F_ConfigPositionEmulation_002();

END_FUNCTION

// ---- 10_Project/11_Emu/10_Config/F_ConfigPositionEmulation_001.TcPOU
FUNCTION F_ConfigPositionEmulation_001








(****************************** 10-001-0201-01-0 ************************************)
(**************************** LowLift Unit Emulation ***************************)
// Configuration emulation
fbF_10_001_0201_01_0_Emulation.Config.Position_Max_Down			:= 0;
fbF_10_001_0201_01_0_Emulation.Config.Position_Max_Up	  			:= 600;	
fbF_10_001_0201_01_0_Emulation.Config.Position_Down				:= 100;
fbF_10_001_0201_01_0_Emulation.Config.Position_Up	  				:= 500;






(****************************** 10-001-0203-02-0 ************************************)
(******************************** Profile Check Emulation *****************************)
// Configuration emulation
fbF_10_001_0203_02_0_Emulation.Config.DefaultWidth					:= 800;
fbF_10_001_0203_02_0_Emulation.Config.DefaultLength					:= 1200;	

(****************************** 10-001-0203-03-0 ************************************)
// Configuration Scanner emulation
fbF_10_001_0203_03_0_Emulation.Config.CreateLabelLength				:= 18; // Label length when ATQ Msg field data is set to 'CREATECODE'







(****************************** 10-001-0204-01-0 ************************************)
(**************************** TurnTable with one drive ***************************)
// Configuration emulation
fbF_10_001_0204_01_0_Emulation.Config.TurnTableCfg.Position_Max_CW	  	:= 500;
fbF_10_001_0204_01_0_Emulation.Config.TurnTableCfg.Position_Max_CCW	:= 0;	
fbF_10_001_0204_01_0_Emulation.Config.TurnTableCfg.Position_CW	  		:= 400;
fbF_10_001_0204_01_0_Emulation.Config.TurnTableCfg.Position_CCW		:= 0;
fbF_10_001_0204_01_0_Emulation.Config.TurnTableCfg.Position_Middle_CW	:= 200;
fbF_10_001_0204_01_0_Emulation.Config.TurnTableCfg.Position_Middle_CCW	:= 200;






(****************************** 10-001-0207-02-0 ************************************)
(****************************** PalletMagazine Addon *************************************)

fbF_10_001_0207_02_0_Emulation.Config.MaxLiftPosition			:= 600;
fbF_10_001_0207_02_0_Emulation.Config.NumberPalletStack		:= 5;	
fbF_10_001_0207_02_0_Emulation.Config.NumberPalletFull			:= 7;






(****************************** 10-001-0209-01-0 ************************************)
(**************************** Transfer Unit Emulation ***************************)
// Configuration emulation
fbF_10_001_0209_01_0_Emulation.Config.Position_Max_Down			:= 0;
fbF_10_001_0209_01_0_Emulation.Config.Position_Max_Up	  			:= 400;	
fbF_10_001_0209_01_0_Emulation.Config.Position_Down				:= 100;
fbF_10_001_0209_01_0_Emulation.Config.Position_Up	  				:= 300;






(****************************** 10-001-0212-01-0 ************************************)
(**************************** Transfer Unit Emulation ***************************)
// Configuration emulation
fbF_10_001_0212_01_0_Emulation.Config.Position_Max_Down			:= 0;
fbF_10_001_0212_01_0_Emulation.Config.Position_Max_Up	  			:= 400;	
fbF_10_001_0212_01_0_Emulation.Config.Position_Down				:= 100;
fbF_10_001_0212_01_0_Emulation.Config.Position_Up	  				:= 300;



(****************************** 10-001-0213-02-0 ************************************)
(****************************** PalletMagazine Addon *************************************)

fbF_10_001_0213_02_0_Emulation.Config.MaxLiftPosition			:= 600;
fbF_10_001_0213_02_0_Emulation.Config.NumberPalletStack		:= 5;	
fbF_10_001_0213_02_0_Emulation.Config.NumberPalletFull			:= 7;





















(****************************** 10-001-0221-01-0 ************************************)
(**************************** Transfer Unit Emulation ***************************)
// Configuration emulation
fbF_10_001_0221_01_0_Emulation.Config.Position_Max_Down			:= 0;
fbF_10_001_0221_01_0_Emulation.Config.Position_Max_Up	  			:= 400;	
fbF_10_001_0221_01_0_Emulation.Config.Position_Down				:= 100;
fbF_10_001_0221_01_0_Emulation.Config.Position_Up	  				:= 300;




(****************************** 10-001-0222-01-0 ************************************)
(**************************** Transfer Unit Emulation ***************************)
// Configuration emulation
fbF_10_001_0222_01_0_Emulation.Config.Position_Max_Down			:= 0;
fbF_10_001_0222_01_0_Emulation.Config.Position_Max_Up	  			:= 400;	
fbF_10_001_0222_01_0_Emulation.Config.Position_Down				:= 100;
fbF_10_001_0222_01_0_Emulation.Config.Position_Up	  				:= 300;










(****************************** 10-001-0230-01-0 ************************************)
(**************************** TransferCC Emulation ***************************)
// Configuration emulation
fbF_10_001_0230_01_0_Emulation.Config.Position_Max_Left			:= 0;
fbF_10_001_0230_01_0_Emulation.Config.Position_Max_Right	  			:= 600;	
fbF_10_001_0230_01_0_Emulation.Config.Position_Left				:= 100;
fbF_10_001_0230_01_0_Emulation.Config.Position_Right	  				:= 500;

END_FUNCTION

// ---- 10_Project/11_Emu/10_Config/F_ConfigPositionEmulation_002.TcPOU
FUNCTION F_ConfigPositionEmulation_002

END_FUNCTION

// ---- 10_Project/11_Emu/10_Config/F_ConfigGroupEmulation.TcPOU
FUNCTION F_ConfigGroupEmulation




(********************************* Group *************************************
 Switching Group  
**********************************************************************************)
fbSG_001_Emulation.Config.Autostart := TRUE;


(********************************* Group *************************************
 Switching Group  
**********************************************************************************)
fbSG_002_Emulation.Config.Autostart := TRUE;

END_FUNCTION

// ---- 10_Project/11_Emu/10_Config/F_ConfigSubSystemEmulation.TcPOU
FUNCTION F_ConfigSubSystemEmulation : BOOL

;

END_FUNCTION

// ---- 10_Project/10_App/11_Custom/F_DebugCompositionCustomization.TcPOU
FUNCTION F_DebugCompositionCustomization : BOOL



(****************************************************************************************
   Add custom code that shall be executed during debug here.
*****************************************************************************************)
;


(****************************************************************************************
   Example: Configure project when running Demo3D simulator
*****************************************************************************************)
IF(DEMO3D_SIM_ENABLED) THEN
	;
	(*
	Groups.fbSG_001.HW_Inputs.AutoOnPB 						:= TRUE;
	Groups.fbSG_001.HW_Inputs.EmergencyCircuitOK 			:= TRUE;
	Groups.fbSG_001.HW_Inputs.ManAutoSW 					:= TRUE;
	Groups.fbSG_001.HW_Inputs.ResetErrorPB 					:= ResetErrorSG1; 
	Groups.fbSG_001.HW_Inputs.MainContactorOFF				:= TRUE; 
	Groups.fbSG_001.HW_Inputs.FeedbackMainContactorOFF[1]	:= TRUE; 
	Groups.fbSG_001.HW_Inputs.FeedbackMainContactorOFF[2]	:= TRUE; 
	Groups.fbSG_001.HW_Inputs.FeedbackMainContactorOFF[3]	:= TRUE; 
	Groups.fbSG_001.HW_Inputs.FeedbackMainContactorOFF[4]	:= TRUE; 
	Groups.fbSG_001.HW_Inputs.FireAlarm						:= TRUE; 
	*)
END_IF

END_FUNCTION

// ---- 20_Product/20_ProBox/22_ProMove/14_Groups/10_App/FB_ProBOXSG.TcPOU
FUNCTION_BLOCK FB_ProBOXSG EXTENDS FB_GroupConv
(**************************************************************************************
 * 	Application		:	BoxControl Framework
 *	Revision		:	$$
 *	Revision date	:	$$
 *	Last changed by	:	$$
 *	URL				:	$$
 *
 *	Purpose			:	ProBox Switching group - Controls a group of elements.
 *
 * ------------------------------------------------------------------------------------
 *	Copyright Swisslog [IP AG], Switzerland. All rights reserved.
 * 
 * ------------------------------------------------------------------------------------
 *	
 * 	Revision History: 
 *
 * 	VERSION			DATE			INITIALS			DESCRIPTION 
 **************************************************************************************)
VAR_INPUT
	HW_Inputs				: ST_HW_InputsSG_ProBOX; // HW-Inputs 
	Config					: ST_CFG_ProBOXSG; // Configuration 
	LocalStopCmd			: BOOL; // Stopping cmd
END_VAR

VAR_OUTPUT
	HW_Outputs				: ST_HW_OutputsSG_ProBOX; // HW-Outputs
	CtrlOut					: ST_CtlrOutProBoxSG; // Summary of input commands from Operator panel(s)
END_VAR

VAR
	ProBoxSG_CFG			: ST_CFG_ProBoxSG;
	Inputs					: ST_SG_Inputs_ProBOX; // Module internal inputs
	Outputs					: ST_SG_Outputs_ProBOX; // Module Internal outputs
	ResetFlag				: BOOL; // Flag to detect reset pulse
	PendingElementError		: BOOL; // An member element is in error state
	fbStartingDelay			: TON; // Timer for startup delay 
	fbForcedStopDelay		: TON; // Timer for forcing a group to stop
	fbResetPulse			: TOF; // Timer for a longer reset pulse
	fbTrigReset				: R_TRIG; // Reset positive flag
	i						: INT;
	ManualModeDelayCnt		: INT; //Delay the Manual Mode  a few cycle in order to send GSR with correct stopped state
END_VAR

VAR PERSISTENT
	Settings				: ST_CFG_ProBoxSG; // Settings - Active configuration
END_VAR

(**************************************************************************************************************
   Input mapping
***************************************************************************************************************)
A_InputMapping();


(**************************************************************************************************************
   Initialization
***************************************************************************************************************)
A_Init();


(**************************************************************************************************************
   Monitoring input signals
***************************************************************************************************************)
A_SignalMonitoring();

//Process Emergency State signal
_M_ProcessEmgState();


(**************************************************************************************************************
   Errorhandler
***************************************************************************************************************)
A_ErrorHandler();


(**************************************************************************************************************
  Mode control
***************************************************************************************************************)
A_ModeControl();


(**************************************************************************************************************
  State control
***************************************************************************************************************)
A_StateControl();


(**************************************************************************************************************
   InterfaceHandlerOut
***************************************************************************************************************)
A_InterfaceHandlerOut();
	

(**************************************************************************************************************
   Output mapping
***************************************************************************************************************)	
A_OutputMapping();

METHOD PRIVATE _M_ProcessEmgState : BOOL
VAR_INST
	InternalStopPending 	: BOOL :=TRUE; //has internal error memory flag
	fbBlink_ExternalStop	: FB_GeneratePulse := (Start := TRUE, PulseTimeOn := T#1S, PulseTimeOff := T#2S); // On 1 sec, off 2 sec
END_VAR
VAR
	InternalStop	: BOOL;
	ExternalStop	: BOOL;
	LampState		: BOOL; //Lamp State
	EmgOk			: BOOL := FALSE;
END_VAR
InternalStop := NOT Inputs.States.EmgStatus.eInternal OR Inputs.States.EmgStatus.eInternError;
ExternalStop := NOT Inputs.States.EmgStatus.eExternal;

IF(NOT GroupData.Init) THEN
	InternalStopPending:=FALSE;
END_IF

//EMG STOP
IF(ExternalStop OR InternalStop) THEN			
	//Internal emg stop is no longer active, but External (safety zone is not acknowledged)	
	IF(ExternalStop AND InternalStopPending AND NOT InternalStop) THEN
		LampState := System.fbBlink_500ms.Pulse;	
	// IF External stop but internal (AK group) is ok
	ELSIF(ExternalStop AND NOT InternalStop) THEN
		fbBlink_ExternalStop();
		LampState := fbBlink_ExternalStop.Pulse;
	ELSE
		LampState := TRUE;
		InternalStopPending := InternalStop; //Set Mem flag
	END_IF

ELSE	
	LampState := FALSE;
	InternalStopPending := FALSE;
	EmgOk:=TRUE;
END_IF


Inputs.States.EmergencyCircuitOK := EmgOk;
Outputs.EmgStopStatus := _M_ProcessEmgState := LampState;
END_METHOD

METHOD PRIVATE _M_ProcessInputs

VAR
	i,j:INT;
	iMax:INT;
END_VAR
	 
//process inputs and create summary
//AK
	Inputs.OpSummary.OpAutoOn		:= HW_Inputs.AK.OpAutoOn;
	Inputs.OpSummary.OpManAuto		:= HW_Inputs.AK.OpManAuto; //NC
	Inputs.OpSummary.OpMcOff 		:= HW_Inputs.AK.OpMcOff; //NC
	Inputs.OpSummary.OpMcOn 		:= HW_Inputs.AK.OpMcOn;
	Inputs.OpSummary.OpResetError	:= HW_Inputs.AK.OpResetError;
	Inputs.OpSummary.OpResetSafety	:= HW_Inputs.AK.OpResetSafety;	
	Inputs.OpSummary.OpEntryReq   	:= HW_Inputs.AK.OpEntryReq; //NC //Hi=Auto, low=Entry
	Inputs.OpSummary.OpEmgDrive   	:= HW_Inputs.AK.OpEmgDrive AND HW_Inputs.AK.OpManAuto = FALSE; (* and Manual mode*)
	FOR j:=1 TO 2 DO
		Inputs.OpSummary.Conv[j].OpDriveCvFwd := HW_Inputs.AK.Conv[j].OpDriveCvFwd AND HW_Inputs.AK.OpManAuto = FALSE; (*Manual mode*) 
		Inputs.OpSummary.Conv[j].OpDriveCvRev := HW_Inputs.AK.Conv[j].OpDriveCvRev AND HW_Inputs.AK.OpManAuto = FALSE; (*Manual mode*)		
		Inputs.OpSummary.Conv[j].OpMovePos 	  := HW_Inputs.AK.Conv[j].OpMovePos    AND HW_Inputs.AK.OpManAuto = FALSE; (*Manual mode*)
		Inputs.OpSummary.Conv[j].OpMoveNeg    := HW_Inputs.AK.Conv[j].OpMoveNeg    AND HW_Inputs.AK.OpManAuto = FALSE; (*Manual mode*)
	END_FOR	
	



//AP
	iMax :=SEL(Settings.NumberOfAPs<GVL_PB_SG.NUMBER_OF_AP_PANELS, GVL_PB_SG.NUMBER_OF_AP_PANELS, Settings.NumberOfAPs);
	FOR i:=1 TO iMax DO 
		Inputs.OpSummary.OpAutoOn		:= Inputs.OpSummary.OpAutoOn 		OR HW_Inputs.AP[i].OpAutoOn;
		Inputs.OpSummary.OpManAuto		:= Inputs.OpSummary.OpManAuto 		AND HW_Inputs.AP[i].OpManAuto; //NC
		Inputs.OpSummary.OpMcOff 		:= Inputs.OpSummary.OpMcOff 		AND HW_Inputs.AP[i].OpMcOff; //NC
		Inputs.OpSummary.OpMcOn 		:= Inputs.OpSummary.OpMcOn			OR HW_Inputs.AP[i].OpMcOn;
		Inputs.OpSummary.OpResetError	:= Inputs.OpSummary.OpResetError 	OR HW_Inputs.AP[i].OpResetError;
		Inputs.OpSummary.OpResetSafety  := Inputs.OpSummary.OpResetSafety 	OR HW_Inputs.AP[i].OpResetSafety;		
		Inputs.OpSummary.OpEntryReq     := Inputs.OpSummary.OpEntryReq     AND HW_Inputs.AP[i].OpEntryReq; //NC, Hi=Auto, low=Entry
		Inputs.OpSummary.OpEmgDrive     := Inputs.OpSummary.OpEmgDrive     OR (HW_Inputs.AP[i].OpEmgDrive    AND HW_Inputs.AP[i].OpManAuto = FALSE); (*Manual mode*)
		// manual controls of the carriage only allowed if switch is in manual mode
		FOR j:=1 TO 2 DO		 
			Inputs.OpSummary.Conv[j].OpDriveCvFwd := Inputs.OpSummary.Conv[j].OpDriveCvFwd OR (HW_Inputs.AP[i].Conv[j].OpDriveCvFwd AND HW_Inputs.AP[i].OpManAuto = FALSE); (*Manual mode*)
			Inputs.OpSummary.Conv[j].OpDriveCvRev := Inputs.OpSummary.Conv[j].OpDriveCvRev OR (HW_Inputs.AP[i].Conv[j].OpDriveCvRev AND HW_Inputs.AP[i].OpManAuto = FALSE); (*Manual mode*)
			Inputs.OpSummary.Conv[j].OpMovePos    := Inputs.OpSummary.Conv[j].OpMovePos    OR (HW_Inputs.AP[i].Conv[j].OpMovePos    AND HW_Inputs.AP[i].OpManAuto = FALSE); (*Manual mode*)
			Inputs.OpSummary.Conv[j].OpMoveNeg    := Inputs.OpSummary.Conv[j].OpMoveNeg    OR (HW_Inputs.AP[i].Conv[j].OpMoveNeg    AND HW_Inputs.AP[i].OpManAuto = FALSE); (*Manual mode*)
		END_FOR	
		
	END_FOR
END_METHOD

ACTION A_ErrorHandler:
(**************************************************************************************
 * 	NAME		A_ErrorHandling
 * 	FUNCTION	Handles group or member errors
 **************************************************************************************)
 

(**************************************************************************************************************
  Monitor group errors
***************************************************************************************************************)
M_MonitorGroupErrors();


(**************************************************************************************************************
  Input group reset
***************************************************************************************************************)

// Reset command
IF Inputs.Command.ResetErrorPB AND NOT ResetFlag THEN
	
	// If a group reset has to reset member elements as well
	IF Settings.ResetMemberElements THEN	

		// Forward reset to memeber elements
		fbGroupManager.M_ResetMemberElements(SettingsGroup.eGroupNumber);
	END_IF
		
	// Reset group itself
	GroupData.ErrorData.Error.ResetError := TRUE;
	
	// Save flag
	ResetFlag := TRUE;
	
// Reset command released
ELSIF NOT Inputs.Command.ResetErrorPB THEN
	// Reset flag
	ResetFlag := FALSE;
END_IF
END_ACTION

ACTION A_Init:
(**************************************************************************************
 * 	NAME		A_Init
 * 	FUNCTION	Initialize Group
 **************************************************************************************)

// Update Registry
M_UpdateRegistry();
 
// Set init flag after one cycle
IF NOT GroupData.Init AND GroupData.InitRunning THEN
	// When subsystem is started and initialization is allowed
	IF GroupData.OperationState.Info.SystemReady AND 
	   SettingsGroup.eGroupNumber < GroupData.OperationState.InitRelease.eLimitGroup THEN
	   
		IF M_InitGroup(FALSE) THEN
			// Group initialized - and initialization done
			GroupData.Init := TRUE;
			GroupData.InitRunning := FALSE;
			
			// Set reset cmd
			GroupData.ErrorData.Error.ResetError := TRUE;
			
			DebugMsg := CONCAT('Initialization done. Group: ', ConfigGroup.GroupName);
			fbDebugMsg.M_SendInfoMsg(DebugMsg);
		END_IF
	END_IF
// If the group is not initialized
ELSIF NOT GroupData.Init THEN
	
	// Reset internal variables
	ResetFlag := FALSE;
	PendingElementError := FALSE;
	fbStartingDelay(IN := FALSE);
	fbForcedStopDelay(IN := FALSE);
	GroupData.OperationState := GroupBase.OperationStateEmpty;
	ITC.Commands.Start := FALSE;
	ITC.Commands.Stop := FALSE;
	ITC.Commands.eMode := E_PositionMode.UNKNOWN_MODE;
	
	// Load group specific configuration to settings
	Settings := Config;
	
	// Reset values and load config
	M_PreInit();
	GroupData.InitRunning := SettingsGroup.eGroupNumber > 0;
END_IF
END_ACTION

ACTION A_InputMapping:
(**************************************************************************************
 * 	NAME		A_InputMapping
 * 	FUNCTION	Input mapping
 **************************************************************************************)
 
 
(**************************************************************************************************************
   Hardware Inputs
***************************************************************************************************************)

//Summarize inputs and set Inputs.OpSummary
_M_ProcessInputs();

// Mode
Inputs.Command.AutoMode   			:= Inputs.OpSummary.OpManAuto;//HW_Inputs.ManAutoSW;
Inputs.Command.ManualMode 			:= NOT Inputs.OpSummary.OpManAuto;

// Control
Inputs.Command.StartPB 				:=Inputs.OpSummary.OpAutoOn; //HW_Inputs.AutoOnPB;
Inputs.Command.StopPB  				:= FALSE;
Inputs.Command.ResetErrorPB			:= Inputs.OpSummary.OpResetError; //HW_Inputs.ResetErrorPB;
Inputs.Command.ResetEmgPB			:= Inputs.OpSummary.OpResetSafety; //HW_Inputs.ResetEmgergencyPB;

// Signal states							   
//Inputs.States.EmergencyCircuitOK 	:= HW_Inputs.EmergencyCircuitOK;

	// Fire alarm
IF Settings.FireAlarmUsed THEN 
	Inputs.States.FireAlarm				:= NOT HW_Inputs.Diag.FireAlarm;
ELSE Inputs.States.FireAlarm			:= FALSE;
END_IF
	
	// Checks all connected Main Contactor feedback							   
FOR i := 1 TO Settings.NumberOfContactors DO
	IF HW_Inputs.Diag.FeedbackMainContactorOFF[i] THEN
		Inputs.States.MainContactorOFF :=TRUE;
		EXIT;
	ELSE
		Inputs.States.MainContactorOFF :=FALSE;
	END_IF
END_FOR

//Inputs.States.MainContactorOFF   	:= HW_Inputs.MainContactorOFF[K.NumberOfContactors];								   

(**************************************************************************************************************
   SubsystemManager states
***************************************************************************************************************)
// Get Subsystem state
M_GetSubsystemStates();

(**************************************************************************************************************
   GroupManager
***************************************************************************************************************)

// Get group member state
Inputs.GroupMemberState 			:= fbGroupManager.M_GetGroupMemberState(SettingsGroup.eGroupNumber);
END_ACTION

ACTION A_InterfaceHandlerOut:
(**************************************************************************************
 * 	NAME		A_InterfaceHandlerOut
 * 	FUNCTION	Handle outgoing interfaces
 **************************************************************************************)
 
 
 (**************************************************************************************************************
   ITC Handler Out
***************************************************************************************************************)
M_ITC_ProcessOut();
END_ACTION

ACTION A_ModeControl:
(**************************************************************************************
 * 	NAME		A_ModeControl
 * 	FUNCTION	Handle group modes
 **************************************************************************************)
 
// Group mode
CASE GroupData.OperationState.eMode OF

	(*******************************************************************************
	  Mode: Unknown 
	********************************************************************************)
	E_PositionMode.UNKNOWN_MODE:
	
		// Group mode is default Off
		GroupData.OperationState.eMode 		:= E_PositionMode.OFF_MODE;

	(*******************************************************************************
	  Mode: OFF
	********************************************************************************)
	E_PositionMode.OFF_MODE:
	
		// If manual mode is set
		IF Inputs.Command.ManualMode THEN
			// Switch to manual mode
			GroupData.OperationState.eMode := E_PositionMode.MANUAL_MODE;
			
		// If semi auto mode is set
		ELSIF Inputs.Command.SemiAutoMode THEN
			// Switch to semi auto mode
			GroupData.OperationState.eMode := E_PositionMode.SEMI_AUTO;
			
		// If auto mode is set
		ELSIF Inputs.Command.AutoMode THEN
			// Switch to auto mode
			GroupData.OperationState.eMode := E_PositionMode.AUTO_MODE;
		END_IF

	(*******************************************************************************
	  Mode: Manual
	********************************************************************************)
	E_PositionMode.MANUAL_MODE:
	
		// If manual - stay
		IF Inputs.Command.ManualMode THEN
			;
		// If semi auto mode is set
		ELSIF Inputs.Command.SemiAutoMode THEN
			// Switch to semi auto mode
			GroupData.OperationState.eMode := E_PositionMode.SEMI_AUTO;
			
			// Send status report
			ITC.Commands.StatusReport := TRUE;
		
		// If auto is set
		ELSIF Inputs.Command.AutoMode THEN
			// Switch mode to "Auto"
			GroupData.OperationState.eMode := E_PositionMode.AUTO_MODE;
			
			// Send status report
			ITC.Commands.StatusReport := TRUE;
		ELSE
			// Switch group off
			GroupData.OperationState.eMode := E_PositionMode.OFF_MODE;
			
			// Send status report
			ITC.Commands.StatusReport := TRUE;
		END_IF
		
	(*******************************************************************************
	  Mode: Auto
	********************************************************************************)
	E_PositionMode.AUTO_MODE:

		// If mode is switched to manual and group state is stopped (not stopping and not started)
		IF Inputs.Command.ManualMode THEN			
			IF(GroupData.OperationState.eState <> E_PositionState.STOPPING AND GroupData.OperationState.eState <> E_PositionState.STARTED) THEN
				ManualModeDelayCnt:=ManualModeDelayCnt+1;
				IF(ManualModeDelayCnt>3) THEN				
					// Switch mode to "Manual"
					GroupData.OperationState.eMode := E_PositionMode.MANUAL_MODE;
					// Send status report
					ITC.Commands.StatusReport := TRUE;
				END_IF
			END_IF
			
		// If semi auto mode is set
		ELSIF Inputs.Command.SemiAutoMode THEN
			// Switch to semi auto mode
			GroupData.OperationState.eMode := E_PositionMode.SEMI_AUTO;
			
			// Send status report
			ITC.Commands.StatusReport := TRUE;
		
		// If auto - stay
		ELSIF Inputs.Command.AutoMode THEN
			ManualModeDelayCnt:=0;
		ELSE
			// Switch group off
			GroupData.OperationState.eMode := E_PositionMode.OFF_MODE;
			
			// Send status report
			ITC.Commands.StatusReport := TRUE;
		END_IF
			
	(*******************************************************************************
	  Mode: Semi Auto
	********************************************************************************)
	E_PositionMode.SEMI_AUTO:
	
		// If manual is set
		IF Inputs.Command.ManualMode THEN
			// Switch mode to "Manual"
			GroupData.OperationState.eMode := E_PositionMode.MANUAL_MODE;
			
			// Send status report
			ITC.Commands.StatusReport := TRUE;
			
		// If semi auto - stay
		ELSIF Inputs.Command.SemiAutoMode THEN
			;
		
		// If auto is set
		ELSIF Inputs.Command.AutoMode THEN
			// Switch mode to "Auto"
			GroupData.OperationState.eMode := E_PositionMode.AUTO_MODE;
			
			// Send status report
			ITC.Commands.StatusReport := TRUE;
		ELSE
			// Switch group off
			GroupData.OperationState.eMode := E_PositionMode.OFF_MODE;
			
			// Send status report
			ITC.Commands.StatusReport := TRUE;
		END_IF
	
(********************************************************************************
	Error case
*********************************************************************************)
ELSE
	// Programming error
	DebugMsg := CONCAT(	'Programming error - Invalid mode: ', 
						INT_TO_STRING(GroupData.OperationState.eMode));
		
	fbDebugMsg.M_SendErrorMsg(DebugMsg);
END_CASE
END_ACTION

ACTION A_OutputMapping:
(**************************************************************************************
 * 	NAME		A_OutputMapping
 * 	FUNCTION	Output mapping
 **************************************************************************************)
 

(**************************************************************************************************************
   Outputs
***************************************************************************************************************)	

// Group starting warning
Outputs.GroupIsStarting := (GroupData.OperationState.eState = E_PositionState.STARTING);

// Group starting or already started
Outputs.GroupStarted := (GroupData.OperationState.eState = E_PositionState.STARTED) OR 
						((GroupData.OperationState.eState = E_PositionState.STARTING) AND fbBlink_500ms.Pulse);

// Group stopping or already stopped
Outputs.GroupStopped := (GroupData.OperationState.eState = E_PositionState.STOPPED) OR 
						((GroupData.OperationState.eState = E_PositionState.STOPPING) AND fbBlink_500ms.Pulse);

// Group or one of its elements is in error state
Outputs.ErrorPending := (GroupData.ErrorData.ElementErrorPending OR 
						(GroupData.ErrorData.Error.ErrorType = E_ErrorType.ERROR) OR
						(GroupData.ErrorData.Error.ErrorType = E_ErrorType.WARNING)) AND fbBlink_500ms.Pulse;

// Reset trigger
fbTrigReset(CLK := Inputs.Command.ResetErrorPB);

// Extend reset pulse
fbResetPulse(IN := fbTrigReset.Q, PT := Settings.tResetPulse);

// Reset pulse				
Outputs.ResetPulse := fbResetPulse.Q;

(**************************************************************************************************************
   Map Ctrl outputs
***************************************************************************************************************)
CtrlOut.OpSummary			:= Inputs.OpSummary; //Summary of Inputs


(**************************************************************************************************************
   Map Hardware outputs
***************************************************************************************************************)

HW_Outputs.GroupIsStarting	:= Outputs.GroupIsStarting;
HW_Outputs.GroupStarted 	:= HW_Outputs.AutoOnLamp := Outputs.GroupStarted;
HW_Outputs.GroupStopped 	:= Outputs.GroupStopped;
HW_Outputs.ErrorPending 	:= Outputs.ErrorPending;
HW_Outputs.ResetPulse  	 	:= Outputs.ResetPulse;
HW_Outputs.MainContactorLamp := NOT Inputs.States.MainContactorOFF;
HW_Outputs.EmergencyLamp	:= Outputs.EmgStopStatus;
END_ACTION

ACTION A_SignalMonitoring:
(**************************************************************************************
 * 	NAME		A_SignalMonitoring
 * 	FUNCTION	Monitoring input signals
 **************************************************************************************)
 
 // Check for error reset 
F_ResetError(Reset := FALSE, ErrorData := GroupData.ErrorData.ErrorDataSet[2]);
F_ResetError(Reset := FALSE, ErrorData := GroupData.ErrorData.ErrorDataSet[3]);
F_ResetError(Reset := FALSE, ErrorData := GroupData.ErrorData.ErrorDataSet[4]);
// Supervision of Emergency circuit
IF NOT Inputs.States.EmergencyCircuitOK THEN
	// Set error
	F_SetError(	
		ErrorType	:= E_ErrorType.ERROR,
		ErrorParam	:= '',
		ErrorMsg	:= E_ErrorConv.EMERGENCY_STOP,
		ErrorData	:= GroupData.ErrorData.ErrorDataSet[1]);
		
ELSE
	// Auto reset
	F_ResetError(
		Reset := Settings.AutoResetEmergencyCircuit, 
		ErrorData := GroupData.ErrorData.ErrorDataSet[1]);
END_IF

// Supervision of main contactor
IF Inputs.States.MainContactorOFF THEN
	// Set error
	F_SetError(	
		ErrorType	:= E_ErrorType.ERROR,
		ErrorParam	:= '',
		ErrorMsg	:= E_ErrorConv.MAIN_CONTACTOR_OFF,
		ErrorData	:= GroupData.ErrorData.ErrorDataSet[2]);
END_IF


// Fire alarm
IF Inputs.States.FireAlarm THEN
	// Set error
	F_SetError(
		ErrorType	:=E_ErrorType.WARNING,
		ErrorParam	:='',
		ErrorMsg 	:=E_ErrorConv.FIRE_ALARM,
		ErrorData	:=GroupData.ErrorData.ErrorDataSet[3]);
END_IF

// Supervision of  circuit breaker
IF NOT HW_Inputs.Diag.SupplyCircuitBreaker THEN
	// Set error
	F_SetError(	
		ErrorType	:= E_ErrorType.ERROR,
		ErrorParam	:= 'Circuit Break error',
		ErrorMsg	:= E_ErrorConv.CONTROL_VOLTAGE,
		ErrorData	:= GroupData.ErrorData.ErrorDataSet[4]);
END_IF

// Supervision of  ASI Device Status
IF HW_Inputs.Diag.ASI_BusConfigError THEN
	// Set error
	F_SetError(	
		ErrorType	:= E_ErrorType.ERROR,
		ErrorParam	:= 'AS-i Bus error on Group',
		ErrorMsg	:= E_ErrorConv.DEVICE_ERROR,
		ErrorData	:= GroupData.ErrorData.ErrorDataSet[4]);
END_IF



//IF Inputs.Command.ResetPB THEN
//	fbGroupManager.M_ResetMemberElements(SettingsGroup.eGroupNumber);
//END_IF
END_ACTION

ACTION A_StateControl:
(**************************************************************************************
 * 	NAME		A_StateControl
 * 	FUNCTION	Handle group states
 **************************************************************************************)

// Check for error reset
F_ResetError(Reset := FALSE, ErrorData := GroupData.ErrorData.ErrorDataSet[5]);

// Check for error reset
F_ResetError(Reset := FALSE, ErrorData := GroupData.ErrorData.ErrorDataSet[3]);
	
// Update system info
GroupData.OperationState.Info := GroupInterface.In.SubsystemState.Info;
GroupData.OperationState.InitRelease := GroupInterface.In.SubsystemState.InitRelease;
	 	 
// Group states
CASE GroupData.OperationState.eState OF

	(*******************************************************************************
	  Unknown State 
	********************************************************************************)
	E_PositionState.UNKNOWN:
	
		// Group state is stopped by default
		GroupData.OperationState.eLastState := GroupData.OperationState.eState;
		GroupData.OperationState.eState 	:= E_PositionState.STOPPED;
		
		// Send status report
		ITC.Commands.StatusReport := TRUE;
		ITC.Commands.Start := FALSE; 
		ITC.Commands.Stop := FALSE; 

	(*******************************************************************************
	  Stopped
	********************************************************************************)
	E_PositionState.STOPPED:
		// Reset
		ITC.Commands.Stop := FALSE;

		// If the current mode is auto
		IF GroupData.OperationState.eMode = E_PositionMode.AUTO_MODE AND
           GroupInterface.In.SubsystemState.eState = E_PositionState.STARTED AND
   		   GroupData.Init THEN
			
			// If no error is pending
			IF GroupData.ErrorData.Error.ErrorType <> E_ErrorType.ERROR THEN
		
				// If a start command is active
				IF Inputs.Command.StartPB OR
				   Inputs.Command.StartStopPB OR
				   ITC.Commands.Start THEN
				   
				   	// Reset start command
					ITC.Commands.Start := FALSE; 
				   
				   	// If no Stop condition is active
					IF NOT Inputs.Command.StopPB AND
					   NOT LocalStopCmd AND
					   NOT Inputs.StopSubsystem THEN
					   
   						// Change state to "Starting"
					  	GroupData.OperationState.eLastState := GroupData.OperationState.eState;
					  	GroupData.OperationState.eState		:= E_PositionState.STARTING;
						
						// Send status report
						ITC.Commands.StatusReport := TRUE;
						
						// Reset startup delay timer
						fbStartingDelay(IN:= FALSE);
				   	END_IF
				END_IF
			END_IF
		ELSE
			// Reset
			ITC.Commands.Start := FALSE; 
		END_IF

		
	(*******************************************************************************
	  Stopping
	********************************************************************************)
	E_PositionState.STOPPING:

		// Run the ForceStop delay timer 
		fbForcedStopDelay(IN := TRUE, PT :=Config.tForcedStopDelay);

		// Send info message
		IF fbForcedStopDelay.Q THEN
			// Set info
			F_SetError(	
				ErrorType	:= E_ErrorType.WARNING,
				ErrorParam	:= '',
				ErrorMsg	:= E_ErrorConv.FST_STOP_AFTER_TIMEOUT,
				ErrorData	:= GroupData.ErrorData.ErrorDataSet[5]);
		END_IF

		// If all member elements have reported "Stopped", Time is up or an error is active
		// Subsystem is stopped
		IF Inputs.GroupMemberState = E_PositionState.STOPPED OR 
		   GroupData.ErrorData.Error.ErrorType = E_ErrorType.ERROR OR 
		   GroupInterface.In.SubsystemState.eState = E_PositionState.STOPPED OR
		   fbForcedStopDelay.Q THEN
		   
			// Reset startup delay timer 
			fbForcedStopDelay(IN := FALSE);
			
			// Change state to "Stopped"
			GroupData.OperationState.eLastState := GroupData.OperationState.eState;
			GroupData.OperationState.eState		:= E_PositionState.STOPPED;
			
			// Send status report
			ITC.Commands.StatusReport := TRUE;
		END_IF
		
		
	(*******************************************************************************
	  Starting
	********************************************************************************)
	E_PositionState.STARTING:

		// Run startup delay timer
		fbStartingDelay(IN := TRUE, PT := Config.tStartupDelay);
	
		// If a stop command occures during starting,
		// mode is not automatic or an error is active
		IF Inputs.Command.StopPB OR
		   LocalStopCmd OR
		   Inputs.StopSubsystem OR
		   ITC.Commands.Stop OR
		   GroupData.ErrorData.Error.ErrorType = E_ErrorType.ERROR OR 
		   GroupInterface.In.SubsystemState.eState <> E_PositionState.STARTED OR
		   GroupData.OperationState.eMode <> E_PositionMode.AUTO_MODE THEN

			// Change state to "Stopped"
			GroupData.OperationState.eLastState := GroupData.OperationState.eState;
			GroupData.OperationState.eState		:= E_PositionState.STOPPED;
			
			// Send status report
			ITC.Commands.StatusReport := TRUE;
			ITC.Commands.Stop := FALSE;

		// If time is up -> Start group
		ELSIF fbStartingDelay.Q THEN

			// Change state to "Started"
			GroupData.OperationState.eLastState := GroupData.OperationState.eState;
			GroupData.OperationState.eState		:= E_PositionState.STARTED;

			// Send status report
			ITC.Commands.StatusReport := TRUE;
		END_IF

		
	(*******************************************************************************
	  Started (Online/active/running)
	********************************************************************************)
	E_PositionState.STARTED:
		// Start
		ITC.Commands.Start := FALSE;
	
		// If an error is active
		IF GroupData.ErrorData.Error.ErrorType = E_ErrorType.ERROR OR
           GroupInterface.In.SubsystemState.eState = E_PositionState.STOPPED THEN
	
			// Change state to "Stopped"
			GroupData.OperationState.eLastState := GroupData.OperationState.eState;
			GroupData.OperationState.eState		:= E_PositionState.STOPPED;
			
			// Send status report
			ITC.Commands.StatusReport := TRUE;
		
		// If a stop command occures during starting
		// or mode is not automatic
		// or Subsystem want to stop
		// or if a fire alarm is triggered 
		// or switching over to manual mode (Introduced with ProBox 1.8)
		ELSIF Inputs.Command.StopPB OR
			  Inputs.Command.ManualMode OR
		      LocalStopCmd OR
		      Inputs.StopSubsystem OR
			  Inputs.States.FireAlarm OR
		      ITC.Commands.Stop OR
			  GroupInterface.In.SubsystemState.eState <> E_PositionState.STARTED OR
		      GroupData.OperationState.eMode <> E_PositionMode.AUTO_MODE THEN

			// Change state to "Stopping"
			GroupData.OperationState.eLastState := GroupData.OperationState.eState;
			GroupData.OperationState.eState		:= E_PositionState.STOPPING;
			
			// Send status report
			ITC.Commands.StatusReport := TRUE;
			
			// Reset forced stop delay timer
			fbForcedStopDelay(IN := FALSE);
			ITC.Commands.Stop := FALSE;
		END_IF
	
		
(********************************************************************************
	Error case
*********************************************************************************)
ELSE
	// Programming error
	DebugMsg := CONCAT(	'Programming error - Invalid state: ', 
					   	INT_TO_STRING(GroupData.OperationState.eState));
		
	fbDebugMsg.M_SendErrorMsg(DebugMsg);
END_CASE
END_ACTION

//get entry req switch from Cabinets. (Entry Req is NC)
METHOD PUBLIC M_GetEntryRequests : BOOL
VAR_Input
	Index:INT; // index 0 = AK, 1..GVL_PB_SG.NUMBER_OF_AP_PANELS = AP panels
END_VAR
VAR	
END_VAR

IF(Index=0) THEN
	M_GetEntryRequests := HW_Inputs.AK.OpEntryReq;
	RETURN;
ELSIF(Index>0 AND Index <= GVL_PB_SG.NUMBER_OF_AP_PANELS) THEN
	M_GetEntryRequests := HW_Inputs.AP[Index].OpEntryReq;
END_IF
END_METHOD

// Reset Safety Needed
METHOD PUBLIC M_SetEmgStatus
VAR_INPUT
	Status : ST_EmgStatus;
END_VAR

Inputs.States.EmgStatus := Status;
END_METHOD

//Set the HW signal that shall be connected to the LED to indicate status to operator, flashing = Pending, True = Active (solid LED), false = no request, LED OFF
METHOD PUBLIC M_SetEntryReqLed
VAR_INPUT
	Index:INT; 		// The current active index of panels, 0 = AK, 1..GVL_PB_SG.NUMBER_OF_AP_PANELS = AP panels
	Pending:BOOL;	// entry request is pending
	Completed:BOOL; // Entry request finilized by MPD (vc or shuttle) 
END_VAR
VAR
	i:INT;
	TempVal	: BOOL;
END_VAR
//Set entry req
//Set output, blink or solid
FOR i:=0 TO GVL_PB_SG.NUMBER_OF_AP_PANELS DO
	
	TempVal := ((M_GetEntryRequests(i)=FALSE (*Switch turned to Entry*)  OR (Index=i AND Pending)) AND fbBlink_500ms.Pulse) OR (Index=i AND Completed);
	
	IF(i=0) THEN //AK
		HW_outputs.AK_EntryReqLed := TempVal;
	ELSE		
		HW_outputs.AP_EntryReqLed[i] := TempVal; 
	END_IF

END_FOR
END_METHOD

//monitor device states.
METHOD M_SetEtherCatError : BOOL
VAR_INPUT
 Index:INT;
END_VAR
VAR_IN_OUT
	SgInput	:ST_HW_InputsSubsystemManager;
END_VAR
F_ResetError(Reset := FALSE, ErrorData :=GroupData.ErrorData.ErrorDataSet[3]);


IF(SgInput.DeviceState[Index]<>8) THEN
// Set error
F_SetError(	
	ErrorType	:= E_ErrorType.ERROR,
	ErrorParam	:= 'EtherCAT-Device Error',
	ErrorMsg	:= E_ErrorConv.DEVICE_ERROR,
	ErrorData	:= GroupData.ErrorData.ErrorDataSet[3]);	
end_if
END_METHOD

END_FUNCTION_BLOCK

// ---- 20_Product/10_BCF/11_Conv/14_Groups/FB_GroupConv.TcPOU
FUNCTION_BLOCK FB_GroupConv EXTENDS FB_BaseObject
(**************************************************************************************
 * 	Application		:	BoxControl Framework
 *	Revision		:	$Revision: 404529 $
 *	Revision date	:	$Date: 2020-11-19 15:59:09 +0100 (tor, 19 nov 2020) $
 *	Last changed by	:	$Author: b7bolm $
 *	URL				:	$URL: http://almscdc.swisslog.com/repo/SWPD/Development/BoxControlFramework/20_Release/trunk/01_Software/BCF/BCF/JumpStart/20_Product/10_App/14_Groups/10_Lib/10_Conv/FB_GroupConv.TcPOU $
 *
 *	Purpose			:	Group.
 *
 * ------------------------------------------------------------------------------------
 *	Copyright Swisslog [IP AG], Switzerland. All rights reserved.
 * 
 * ------------------------------------------------------------------------------------
 *	
 * 	Revision History: 
 *
 * 	VERSION			DATE			INITIALS			DESCRIPTION
 *	0.1				01.01.2001		swl					Example
 *
 **************************************************************************************)
VAR_INPUT
	ConfigGroup				: ST_CFG_Group; // Base group configuration 
END_VAR

VAR
	GroupBase				: ST_GroupBase; // Summary of variables used from framework
END_VAR

VAR PERSISTENT
	ITC						: ST_ITC_Group; // Internal ITC			
	GroupData				: ST_GroupData; // General data 
	GroupInterface			: ST_GroupInterface; // Group interface
	SettingsGroup			: ST_CFG_Group; // Base group settings 
END_VAR

(**************************************************************************************************************
   Base group - Body is never called!
***************************************************************************************************************)
;

METHOD PROTECTED M_GetSubsystemStates 
(**************************************************************************************
 * 	Application		:	BoxControl Framework
 *	Revision		:	$Revision: 404529 $
 *	Revision date	:	$Date: 2020-11-19 15:59:09 +0100 (tor, 19 nov 2020) $
 *	Last changed by	:	$Author: b7bolm $
 *	URL				:	$URL: http://almscdc.swisslog.com/repo/SWPD/Development/BoxControlFramework/20_Release/trunk/01_Software/BCF/BCF/JumpStart/20_Product/10_App/14_Groups/10_Lib/10_Conv/FB_GroupConv.TcPOU $
 *
 *	Purpose			:	Get states of corresponding subsystem
 *
 * ------------------------------------------------------------------------------------
 *	Copyright Swisslog [IP AG], Switzerland. All rights reserved.
 * 
 * ------------------------------------------------------------------------------------
 *	
 * 	Revision History: 
 *
 * 	VERSION			DATE			INITIALS			DESCRIPTION
 *	0.1				01.01.2001		swl					Example
 *
 **************************************************************************************)
VAR
	mIdx					: INT; // Iterator
	eElementNumber			: E_ElementNumber; 
END_VAR
// Check element is initialized and has valid references
IF __ISVALIDREF(SubsystemRegistry.rSubsystemData) AND
  F_IsSubsystemInitialized() THEN
	// Return 
	GroupInterface.In.SubsystemState := SubsystemRegistry.rSubsystemData.OperationState;
ELSE
	GroupInterface.In.SubsystemState := GroupBase.OperationStateEmpty;
END_IF
END_METHOD

METHOD M_InitGroup : BOOL
(**************************************************************************************
 * 	Application		:	BoxControl Framework
 *	Revision		:	$Revision: 404529 $
 *	Revision date	:	$Date: 2020-11-19 15:59:09 +0100 (tor, 19 nov 2020) $
 *	Last changed by	:	$Author: b7bolm $
 *	URL				:	$URL: http://almscdc.swisslog.com/repo/SWPD/Development/BoxControlFramework/20_Release/trunk/01_Software/BCF/BCF/JumpStart/20_Product/10_App/14_Groups/10_Lib/10_Conv/FB_GroupConv.TcPOU $
 *
 *	Purpose			:	Initialize base functionality of group.
 *
 * ------------------------------------------------------------------------------------
 *	Copyright Swisslog [IP AG], Switzerland. All rights reserved.
 * 
 * ------------------------------------------------------------------------------------
 *	
 * 	Revision History: 
 *
 * 	VERSION			DATE			INITIALS			DESCRIPTION
 *	0.1				01.01.2001		swl					Example
 *
 **************************************************************************************)
 VAR_INPUT
	 mReset		: BOOL; // Force initialization
 END_VAR
 VAR
	 mName		: T_MaxString; // Name with alpha numeric signs only
 END_VAR

// If the init command was an external command
IF mReset THEN
	// Inform the bottom group to initialize
	GroupData.Init := FALSE;
	// Reset values and load config
	M_PreInit();
ELSE
	// Load basic configuration to settings
	SettingsGroup := ConfigGroup;
	
	// Remove non alpha numeric signs
	mName := F_ReduceToAlphaNumeric(InputString := SettingsGroup.GroupName);

	// Update Registry reference with HashCode
	GroupRegistry[SettingsGroup.eGroupNumber].HashCode := F_CreateHashCode(mName);
	
	// Update Registry reference with name
	GroupRegistry[SettingsGroup.eGroupNumber].GroupName := SettingsGroup.GroupName;
	
	// Base group initialized
	M_InitGroup := TRUE;
END_IF
END_METHOD

METHOD PRIVATE M_ITC_GCQ : BOOL
VAR_INPUT
	meChannelSrc		: E_MFCS_CHANNEL; // Number of the source 
	mpData				: PVOID; // Data  pointer 
	mLen				: UDINT; // Data length
END_VAR
// Map data
F_BlockCopy(
	pSrc:= mpData, 
	LenSrc:= mLen, 
	pDest:= ADR(GroupBase.GCQ), 
	LenDest:= SIZEOF(GroupBase.GCQ));
	
// Validate control code
CASE GroupBase.GCQ.Code OF
	(*******************************************************************************
		No code
	********************************************************************************)
	E_ITC_GroupControlCode.NO_CODE:
		// No code received
		;
		
	(*******************************************************************************
		Reset error
	********************************************************************************)
	E_ITC_GroupControlCode.RESET_ERROR:
		// Reset group
		GroupData.ErrorData.Error.ResetError := TRUE;
			
	(*******************************************************************************
		Change state
	********************************************************************************)
	E_ITC_GroupControlCode.CHANGE_STATE:
		// If a command to start was received
		IF GroupBase.GCQ.Variable = 1 THEN
			// Set ITC command start
			ITC.Commands.Start := TRUE;
		
		// If a command to stop was received
		ELSIF GroupBase.GCQ.Variable = 0 THEN
			// Set ITC command stop
			ITC.Commands.Stop := TRUE;
		ELSE
			// Invalid change state received
			DebugMsg := CONCAT('M_ITC_HandleBufferMessages  - Invalid change state', DINT_TO_STRING(GroupBase.GCQ.Variable));
			fbDebugMsg.M_SendErrorMsg(mMessage := DebugMsg);
		END_IF

	(*******************************************************************************
		Change mode
	********************************************************************************)
	E_ITC_GroupControlCode.CHANGE_MODE:
		// Store command to change mode
		ITC.Commands.eMode := DINT_TO_INT(GroupBase.GCQ.Variable);
	
	(*******************************************************************************
		Set Variable
	********************************************************************************)
	E_ITC_GroupControlCode.SET_VARIABLE:
		// Store variable
		ITC.Variable := GroupBase.GCQ.Variable;
	
ELSE
	// Unrecognised ControlRequest message received 
	DebugMsg := CONCAT('M_ITC_HandleBufferMessages - Unknown control code received: ', INT_TO_STRING(GroupBase.GCQ.Code));
	fbDebugMsg.M_SendErrorMsg(mMessage := DebugMsg);
END_CASE

F_ITC_SendGCR(
	eChannelSrc	:= meChannelSrc, 
	GroupName	:= F_ReduceToAlphaNumeric(SettingsGroup.GroupName), 
	Code		:= GroupBase.GCQ.Code, 
	Variable	:= GroupBase.GCQ.Variable, 
	eReturnCode	:= E_ErrorConv.NO_ERROR_CODE);
END_METHOD

METHOD PRIVATE M_ITC_GSQ : BOOL
VAR_INPUT
	meChannelSrc		: E_MFCS_CHANNEL; // Number of the source 
	mpData				: PVOID; // Data  pointer 
	mLen				: UDINT; // Data length
END_VAR
// Map data
F_BlockCopy(
	pSrc:= mpData, 
	LenSrc:= mLen, 
	pDest:= ADR(GroupBase.GSQ), 
	LenDest:= SIZEOF(GroupBase.GSQ));

F_ITC_SendGSR(
	eChannelSrc			:= meChannelSrc, 
	GroupName			:= F_ReduceToAlphaNumeric(SettingsGroup.GroupName), 
	eMode				:= GroupData.OperationState.eMode, 
	eState				:= GroupData.OperationState.eState, 
	eErrorState			:= GroupData.ErrorData.ErrorState, 
	eErrorCode			:= GroupData.ErrorData.Error.ErrorCode.Conv, 
	eErrorType			:= GroupData.ErrorData.Error.ErrorType, 
	ErrorInformation	:= GroupData.ErrorData.Error.ErrorParam, 
	Variable			:= ITC.Variable, 
	eReturnCode			:= E_ErrorConv.NO_ERROR_CODE);
END_METHOD

METHOD M_ITC_ProcessMsg : BOOL
(**************************************************************************************
 * 	Application		:	BoxControl Framework
 *	Revision		:	$Revision: 404529 $
 *	Revision date	:	$Date: 2020-11-19 15:59:09 +0100 (tor, 19 nov 2020) $
 *	Last changed by	:	$Author: b7bolm $
 *	URL				:	$URL: http://almscdc.swisslog.com/repo/SWPD/Development/BoxControlFramework/20_Release/trunk/01_Software/BCF/BCF/JumpStart/20_Product/10_App/14_Groups/10_Lib/10_Conv/FB_GroupConv.TcPOU $
 *
 *	Purpose			:	Handle incoming group ITC messages.
 *
 * ------------------------------------------------------------------------------------
 *	Copyright Swisslog [IP AG], Switzerland. All rights reserved.
 * 
 * ------------------------------------------------------------------------------------
 *	
 * 	Revision History: 
 *
 * 	VERSION			DATE			INITIALS			DESCRIPTION
 *	0.1				01.01.2001		swl					Example
 *
 **************************************************************************************)
VAR_INPUT
	meChannelSrc		: E_MFCS_CHANNEL; // Number of the source 
	mMsgType			: INT; // Message type
	mpData				: PVOID; // Data  pointer 
	mLen				: UDINT; // Data length
END_VAR

// Initialize ITC commands
ITC.Commands.Start 	:= FALSE;
ITC.Commands.Stop 	:= FALSE;
M_ITC_ProcessMsg := TRUE;

// Validate inputs
IF mpData > 0 AND
   mLen > 0 THEN
	// Map enum
	GroupBase.eMsgType := mMsgType;

	// Validate message type
	CASE GroupBase.eMsgType OF
		(*******************************************************************************
		  Status request message
		********************************************************************************)
		E_ITC_MsgTypeConv.GROUP_STATUS_REQUEST:
			M_ITC_GSQ(meChannelSrc := meChannelSrc, mpData := mpData, mLen := mLen);

		(*******************************************************************************
		  Control request message
		********************************************************************************)
		E_ITC_MsgTypeConv.GROUP_CONTROL_REQUEST:
			M_ITC_GCQ(meChannelSrc := meChannelSrc, mpData := mpData, mLen := mLen);
						
		(*******************************************************************************
		  Data Aquisition Request 
		********************************************************************************)
		E_ITC_MsgTypeConv.DATA_ACQUISITION_REQUEST:
			M_ITC_DAQ(meChannelSrc := meChannelSrc, mpData := mpData, mLen := mLen);
		
		(*******************************************************************************
		  Gathered Data Request 
		********************************************************************************)
		E_ITC_MsgTypeConv.GATHERED_DATA_REQUEST:
			M_ITC_GDQ(meChannelSrc := meChannelSrc, mpData := mpData, mLen := mLen);
			
		(*******************************************************************************
		  Visualization information request
		********************************************************************************)			
		E_ITC_MsgTypeConv.VISUALIZATION_INFORMATION_REQUEST:
			M_ITC_VIQ(meChannelSrc := meChannelSrc, mpData := mpData, mLen := mLen);
				

	ELSE
		// Unknown ITC message type received
		DebugMsg := CONCAT('M_ITC_HandleBufferMessages - Unknown message type received: ', INT_TO_STRING(mMsgType));
		fbDebugMsg.M_SendErrorMsg(mMessage := DebugMsg);
	END_CASE
END_IF
END_METHOD

METHOD PROTECTED M_ITC_ProcessOut : BOOL
(**************************************************************************************
 * 	Application		:	BoxControl Framework
 *	Revision		:	$Revision: 404529 $
 *	Revision date	:	$Date: 2020-11-19 15:59:09 +0100 (tor, 19 nov 2020) $
 *	Last changed by	:	$Author: b7bolm $
 *	URL				:	$URL: http://almscdc.swisslog.com/repo/SWPD/Development/BoxControlFramework/20_Release/trunk/01_Software/BCF/BCF/JumpStart/20_Product/10_App/14_Groups/10_Lib/10_Conv/FB_GroupConv.TcPOU $
 *
 *	Purpose			:	Group ITC out interface
 *						Handles internally set ITC commands.
 *
 * ------------------------------------------------------------------------------------
 *	Copyright Swisslog [IP AG], Switzerland. All rights reserved.
 * 
 * ------------------------------------------------------------------------------------
 *	
 * 	Revision History: 
 *
 * 	VERSION			DATE			INITIALS			DESCRIPTION
 *	0.1				01.01.2001		swl					Example
 *
 **************************************************************************************)
VAR
	mNoError			: BOOL; // No error during processing
END_VAR

(*******************************************************************************
	Status Report 
********************************************************************************)
// If a time request request is active
IF ITC.Commands.StatusReport THEN
	
	mNoError := F_ITC_SendGSR(
					eChannelSrc			:= 0, 
					GroupName			:= F_ReduceToAlphaNumeric(SettingsGroup.GroupName), 
					eMode				:= GroupData.OperationState.eMode, 
					eState				:= GroupData.OperationState.eState, 
					eErrorState			:= GroupData.ErrorData.ErrorState, 
					eErrorCode			:= GroupData.ErrorData.Error.ErrorCode.Conv, 
					eErrorType			:= GroupData.ErrorData.Error.ErrorType, 
					ErrorInformation	:= GroupData.ErrorData.Error.ErrorParam, 
					Variable			:= ITC.Variable, 
					eReturnCode			:= E_ErrorConv.NO_ERROR_CODE);
	
	// If sending was successfull
	IF mNoError THEN
		// Reset flag
		ITC.Commands.StatusReport := FALSE;
	ELSE
		// Sending failed
		DebugMsg := 'M_ITC_ProcessOut - Forwarding status report to ITC manager failed.';
		fbDebugMsg.M_SendErrorMsg(mMessage := DebugMsg);
	END_IF
END_IF

(*******************************************************************************
	Status report: No error  
********************************************************************************)
// If a time request request is active
IF ITC.Commands.NoErrorReport THEN
	
	mNoError := F_ITC_SendGSR(
					eChannelSrc			:= 0, 
					GroupName			:= F_ReduceToAlphaNumeric(SettingsGroup.GroupName), 
					eMode				:= GroupData.OperationState.eMode, 
					eState				:= GroupData.OperationState.eState, 
					eErrorState			:= E_ErrorState.OPERATIONAL, 
					eErrorCode			:= E_ErrorConv.NO_ERROR_CODE, 
					eErrorType			:= E_ErrorType.NO_ERROR_PENDING, 
					ErrorInformation	:= '', 
					Variable			:= ITC.Variable, 
					eReturnCode			:= E_ErrorConv.NO_ERROR_CODE);
	
	// If sending was successfull
	IF mNoError THEN
		// Reset flag
		ITC.Commands.NoErrorReport := FALSE;
	ELSE
		// Sending failed
		DebugMsg := 'M_ITC_ProcessOut - Forwarding status report to ITC manager failed.';
		fbDebugMsg.M_SendErrorMsg(mMessage := DebugMsg);
	END_IF
END_IF


(*******************************************************************************
	Control Report 
********************************************************************************)
// If a control report msg request is active
IF ITC.Commands.ControlReport THEN

	mNoError := F_ITC_SendGCR(
					eChannelSrc	:= 0, 
					GroupName	:= F_ReduceToAlphaNumeric(SettingsGroup.GroupName), 
					Code		:= 0, 
					Variable	:= ITC.Variable, 
					eReturnCode	:= E_ErrorConv.NO_ERROR_CODE);

	// If sending was successfull
	IF mNoError THEN
		// Reset flag
		ITC.Commands.ControlReport := FALSE;
	ELSE
		// Sending failed
		DebugMsg := 'M_ITC_ProcessOut - Forwarding control report to ITC manager failed.';
		fbDebugMsg.M_SendErrorMsg(mMessage := DebugMsg);
	END_IF
END_IF
END_METHOD

///Monitor group errors
METHOD PROTECTED M_MonitorGroupErrors : BOOL
(**************************************************************************************
 * Application   : BoxControl Framework
 * Revision date : $Date: 2020-11-19 15:59:09 +0100 (tor, 19 nov 2020) $
 * Author        : CDC
 * ------------------------------------------------------------------------------------
 * © Swisslog AG * Swisslog is not liable for any usage of this source code that is not agreed
 * on between Swisslog and the other party. The mandatory legal liability remains * unaffected.
 * ------------------------------------------------------------------------------------
 * Project revision history:
 *
 * VERSION DATE         INITIALS     DESCRIPTION
 * 0.0     DD.MM.YYYY   name       	 explain customized modifications
 *
 **************************************************************************************)
VAR
	mDataSetIdx				: INT; // Temporary data set index
	mIdx					: INT; // Iterator
END_VAR

(**************************************************************************************************************
   Group error handling
***************************************************************************************************************)

// Store current data set index
mDataSetIdx := GroupData.ErrorData.DataSetIdx;

// Check if an error is stored
IF mDataSetIdx > 0 THEN
	
	// If error type has changed - its gone or type has changed
	IF GroupData.ErrorData.ErrorDataSet[mDataSetIdx].ErrorType <> 
	   GroupData.ErrorData.Error.ErrorType THEN
		
		// If the stored error type was "ERROR"
		IF GroupData.ErrorData.Error.ErrorType = E_ErrorType.ERROR
		   OR GroupData.ErrorData.Error.ErrorType = E_ErrorType.WARNING THEN
			// Send error is gone
			ITC.Commands.NoErrorReport := TRUE;
		END_IF
		
		// Reset stored data index
		GroupData.ErrorData.DataSetIdx := 0;		
				
		// Reset Message
		GroupData.ErrorData.Error.ResetError 		:= FALSE;
		GroupData.ErrorData.Error.ErrorType 		:= NO_ERROR_PENDING;
		GroupData.ErrorData.Error.ErrorCode.Conv 	:= E_ErrorConv.NO_ERROR_CODE;
		GroupData.ErrorData.Error.ErrorParam 		:= '';
	END_IF
	
// Check if an external error is stored
ELSIF GroupData.ErrorData.ExternalError.ErrorType > E_ErrorType.NO_ERROR_PENDING THEN
	// If error type has changed - its gone or type has changed
	IF GroupData.ErrorData.ExternalError.ErrorType <> 
	   GroupData.ErrorData.Error.ErrorType THEN
	   
		// If the stored error type was "ERROR"
		IF GroupData.ErrorData.Error.ErrorType = E_ErrorType.ERROR
		   OR GroupData.ErrorData.Error.ErrorType = E_ErrorType.WARNING THEN
			// Send error is gone
			ITC.Commands.NoErrorReport := TRUE;
		END_IF
		
		// Reset Message
		GroupData.ErrorData.Error.ResetError 	:= FALSE;
		GroupData.ErrorData.Error.ErrorType 	:= NO_ERROR_PENDING;
		GroupData.ErrorData.Error.ErrorCode.Conv:= E_ErrorConv.NO_ERROR_CODE;
		GroupData.ErrorData.Error.ErrorParam 	:= '';
	END_IF
END_IF
	
(**************************************************************************************************************
   Check for new or higher prioritized message
***************************************************************************************************************)
// Loop trough all errors 
FOR mIdx := 1 TO NUMBER_OF_ERROR_SETS DO
	// Detect new or higher prioritized error message
	IF GroupData.ErrorData.ErrorDataSet[mIdx].ErrorType > 
	   GroupData.ErrorData.Error.ErrorType THEN
		
		// Store index of current data set
		GroupData.ErrorData.DataSetIdx := mIdx;
		
		// Update error
		GroupData.ErrorData.Error.ErrorCode.Conv := GroupData.ErrorData.ErrorDataSet[mIdx].ErrorCode.Conv;
		GroupData.ErrorData.Error.ErrorParam := GroupData.ErrorData.ErrorDataSet[mIdx].ErrorParam;
		GroupData.ErrorData.Error.ErrorType := GroupData.ErrorData.ErrorDataSet[mIdx].ErrorType;
		
		// Send Report
		ITC.Commands.StatusReport := TRUE;
	END_IF
	
	// Check is an error is ongoing and a reset command is set
	IF GroupData.ErrorData.Error.ResetError AND 
       GroupData.ErrorData.ErrorDataSet[mIdx].ErrorType <> NO_ERROR_PENDING THEN
	   
		// Reset current error data set
		GroupData.ErrorData.ErrorDataSet[mIdx].ResetError := TRUE;
	END_IF
END_FOR

// Check external error slot
IF GroupData.ErrorData.ExternalError.ErrorType > GroupData.ErrorData.Error.ErrorType THEN

	// Reset lower prioritized previous errors
	mDataSetIdx := 0;
	
	// Update error
	GroupData.ErrorData.Error.ErrorCode.Conv := GroupData.ErrorData.ExternalError.ErrorCode.Conv;
	GroupData.ErrorData.Error.ErrorParam := GroupData.ErrorData.ExternalError.ErrorParam;
	GroupData.ErrorData.Error.ErrorType := GroupData.ErrorData.ExternalError.ErrorType;

	// Send Report
	ITC.Commands.StatusReport := TRUE;
END_IF

// Check is an external error is ongoing and a reset command is set
IF GroupData.ErrorData.Error.ResetError AND 
   GroupData.ErrorData.ExternalError.ErrorType <> NO_ERROR_PENDING THEN
   
	// Reset current error data set
	GroupData.ErrorData.ExternalError.ResetError := TRUE;
END_IF

// If reset command is set
IF GroupData.ErrorData.Error.ResetError THEN
	
	// If the stored error type was "ERROR"
	IF GroupData.ErrorData.Error.ErrorType = E_ErrorType.ERROR THEN
		// Send error is gone
		ITC.Commands.NoErrorReport := TRUE;
	END_IF
	
	// Reset stored data index
	GroupData.ErrorData.DataSetIdx := 0;	

	// Reset Message
	GroupData.ErrorData.Error.ResetError 		:= FALSE;
	GroupData.ErrorData.Error.ErrorType 		:= NO_ERROR_PENDING;
	GroupData.ErrorData.Error.ErrorCode.Conv 	:= E_ErrorConv.NO_ERROR_CODE;
	GroupData.ErrorData.Error.ErrorParam 		:= '';
END_IF

(**************************************************************************************************************
   Group error state
***************************************************************************************************************)

// If group is in error state
IF GroupData.ErrorData.Error.ErrorType = E_ErrorType.ERROR THEN
	// Set error state - ERROR
	GroupData.ErrorData.ErrorState := E_ErrorState.ERROR;
	
// If group is in warning state
ELSIF GroupData.ErrorData.Error.ErrorType = E_ErrorType.WARNING THEN
	// Set error state - WARNING
	GroupData.ErrorData.ErrorState := E_ErrorState.WARNING;

// If group has no error or an info is pending
ELSIF GroupData.ErrorData.Error.ErrorType = E_ErrorType.NO_ERROR_PENDING OR 
	  GroupData.ErrorData.Error.ErrorType = E_ErrorType.INFO  THEN
	// Set error state - Operational
	GroupData.ErrorData.ErrorState := E_ErrorState.OPERATIONAL;

ELSE
	// Otherwise -> Unknown
	GroupData.ErrorData.ErrorState := E_ErrorState.UNKNOWN;
END_IF

(**************************************************************************************************************
   Monitor elements
***************************************************************************************************************)
GroupData.ErrorData.ElementErrorPending := fbGroupManager.M_GroupMemberErrorPending(SettingsGroup.eGroupNumber);
END_METHOD

METHOD M_PreInit : BOOL
(**************************************************************************************
 * 	Application		:	BoxControl Framework
 *	Revision		:	$Revision: 404529 $
 *	Revision date	:	$Date: 2020-11-19 15:59:09 +0100 (tor, 19 nov 2020) $
 *	Last changed by	:	$Author: b7bolm $
 *	URL				:	$URL: http://almscdc.swisslog.com/repo/SWPD/Development/BoxControlFramework/20_Release/trunk/01_Software/BCF/BCF/JumpStart/20_Product/10_App/14_Groups/10_Lib/10_Conv/FB_GroupConv.TcPOU $
 *
 *	Purpose			:	Preinitialize 
 *						Clears values and load settings
 *
 * ------------------------------------------------------------------------------------
 *	Copyright Swisslog [IP AG], Switzerland. All rights reserved.
 * 
 * ------------------------------------------------------------------------------------
 *	
 * 	Revision History: 
 *
 * 	VERSION			DATE			INITIALS			DESCRIPTION
 *	0.1				01.01.2001		swl					Example
 *
 **************************************************************************************)
VAR
END_VAR
(**************************************************************************************
	Load number to identify
***************************************************************************************)
SettingsGroup := ConfigGroup;
END_METHOD

METHOD M_ResetError : BOOL
(**************************************************************************************
 * 	Application		:	BoxControl Framework
 *	Revision		:	$Revision: 404529 $
 *	Revision date	:	$Date: 2020-11-19 15:59:09 +0100 (tor, 19 nov 2020) $
 *	Last changed by	:	$Author: b7bolm $
 *	URL				:	$URL: http://almscdc.swisslog.com/repo/SWPD/Development/BoxControlFramework/20_Release/trunk/01_Software/BCF/BCF/JumpStart/20_Product/10_App/14_Groups/10_Lib/10_Conv/FB_GroupConv.TcPOU $
 *
 *	Purpose			:	Reset group errors.
 *
 * ------------------------------------------------------------------------------------
 *	Copyright Swisslog [IP AG], Switzerland. All rights reserved.
 * 
 * ------------------------------------------------------------------------------------
 *	
 * 	Revision History: 
 *
 * 	VERSION			DATE			INITIALS			DESCRIPTION
 *	0.1				01.01.2001		swl					Example
 *
 **************************************************************************************)
// If the group is in error
IF GroupData.ErrorData.Error.ErrorType  <> E_ErrorType.NO_ERROR_PENDING  THEN
	// Send reset
	GroupData.ErrorData.Error.ResetError := TRUE;
END_IF

M_ResetError := TRUE;
END_METHOD

METHOD M_ResetExternalError : BOOL
(**************************************************************************************
 * 	Application		:	BoxControl Framework
 *	Revision		:	$Revision: 404529 $
 *	Revision date	:	$Date: 2020-11-19 15:59:09 +0100 (tor, 19 nov 2020) $
 *	Last changed by	:	$Author: b7bolm $
 *	URL				:	$URL: http://almscdc.swisslog.com/repo/SWPD/Development/BoxControlFramework/20_Release/trunk/01_Software/BCF/BCF/JumpStart/20_Product/10_App/14_Groups/10_Lib/10_Conv/FB_GroupConv.TcPOU $
 *
 *	Purpose			:	Reset external error
 *						
 *
 * ------------------------------------------------------------------------------------
 *	Copyright Swisslog [IP AG], Switzerland. All rights reserved.
 * 
 * ------------------------------------------------------------------------------------
 *	
 * 	Revision History: 
 *
 * 	VERSION			DATE			INITIALS			DESCRIPTION
 *	0.1				01.01.2001		swl					Example
 *
 **************************************************************************************)
 VAR_INPUT
	mReset		: BOOL; // Force reset
END_VAR
// Initialize
M_ResetExternalError := FALSE;

// Reset error if ResetError command or reset command is set 
IF GroupData.ErrorData.ExternalError.ResetError OR mReset THEN
	// Clear error
	GroupData.ErrorData.ExternalError.ResetError 		:= FALSE; 
	GroupData.ErrorData.ExternalError.ErrorType 		:= NO_ERROR_PENDING;
	GroupData.ErrorData.ExternalError.ErrorCode.Conv	:= E_ErrorConv.NO_ERROR_CODE;
	GroupData.ErrorData.ExternalError.ErrorParam 		:= '';
	M_ResetExternalError 								:= TRUE;
END_IF
END_METHOD

METHOD M_SetExternalError : BOOL
(**************************************************************************************
 * 	Application		:	BoxControl Framework
 *	Revision		:	$Revision: 404529 $
 *	Revision date	:	$Date: 2020-11-19 15:59:09 +0100 (tor, 19 nov 2020) $
 *	Last changed by	:	$Author: b7bolm $
 *	URL				:	$URL: http://almscdc.swisslog.com/repo/SWPD/Development/BoxControlFramework/20_Release/trunk/01_Software/BCF/BCF/JumpStart/20_Product/10_App/14_Groups/10_Lib/10_Conv/FB_GroupConv.TcPOU $
 *
 *	Purpose			:	Set error
 *						Wrapped to a function to improve debugging and readability.
 *						
 *
 * ------------------------------------------------------------------------------------
 *	Copyright Swisslog [IP AG], Switzerland. All rights reserved.
 * 
 * ------------------------------------------------------------------------------------
 *	
 * 	Revision History: 
 *
 * 	VERSION			DATE			INITIALS			DESCRIPTION
 *	0.1				01.01.2001		swl					Example
 *
 **************************************************************************************)
 VAR_INPUT
	mErrorType		: E_ErrorType; // Error message type
	mErrorParam		: STRING(System.ERROR_PARAM_STRINGLENGTH); // Error parameter
	mErrorCode		: INT; // Error message
END_VAR
// Initialize
M_SetExternalError := FALSE;

// Check that the values are valid
IF mErrorType > E_ErrorType.NO_ERROR_PENDING AND mErrorCode > E_ErrorConv.NO_ERROR_CODE THEN

	GroupData.ErrorData.ExternalError.ErrorCode.Conv := mErrorCode;
	GroupData.ErrorData.ExternalError.ErrorType := mErrorType;
	GroupData.ErrorData.ExternalError.ErrorParam := mErrorParam;

	M_SetExternalError := TRUE;
END_IF
END_METHOD

METHOD M_UpdateRegistry
(**************************************************************************************
 * 	Application		:	BoxControl Framework
 *	Revision		:	$Revision: 404529 $
 *	Revision date	:	$Date: 2020-11-19 15:59:09 +0100 (tor, 19 nov 2020) $
 *	Last changed by	:	$Author: b7bolm $
 *	URL				:	$URL: http://almscdc.swisslog.com/repo/SWPD/Development/BoxControlFramework/20_Release/trunk/01_Software/BCF/BCF/JumpStart/20_Product/10_App/14_Groups/10_Lib/10_Conv/FB_GroupConv.TcPOU $
 *
 *	Purpose			:	Update registry information
 *
 * ------------------------------------------------------------------------------------
 *	Copyright Swisslog [IP AG], Switzerland. All rights reserved.
 * 
 * ------------------------------------------------------------------------------------
 *	
 * 	Revision History: 
 *
 * 	VERSION			DATE			INITIALS			DESCRIPTION
 *	0.1				01.01.2001		swl					Example
 *
 **************************************************************************************)
VAR_INPUT
END_VAR
VAR
	mIdx	: INT;
END_VAR

IF ConfigGroup.eGroupNumber > E_GroupNumber.G_BEGIN_GROUP THEN

	GroupRegistry[ConfigGroup.eGroupNumber].rGroupData REF= GroupData;
	GroupRegistry[ConfigGroup.eGroupNumber].rGroupInterface REF= GroupInterface;
	GroupRegistry[ConfigGroup.eGroupNumber].rSettingsGroup REF= SettingsGroup;
END_IF
END_METHOD

END_FUNCTION_BLOCK

// ---- 20_Product/10_BCF/11_Conv/15_Subsystem/10_Helper/F_IsSubsystemInitialized.TcPOU
FUNCTION F_IsSubsystemInitialized : BOOL
(**************************************************************************************
 * 	Application		:	BoxControl Framework
 *	Revision		:	$Revision: 404529 $
 *	Revision date	:	$Date: 2018-04-23 08:21:38 +0200 (Mo., 23 Apr 2018) $
 *	Last changed by	:	$Author: b7bolm $
 *	URL				:	$URL: http://almscdc.swisslog.com/repo/SWPD/Development/BoxControlFramework/20_Release/trunk/01_Software/BCF/BCF/JumpStart/20_Product/10_App/15_Subsystem/10_Lib/10_Conv/10_Functions/F_IsSubsystemInitialized.TcPOU $
 *
 *	Purpose			:	Returns group base data
 *
 * ------------------------------------------------------------------------------------
 *	Copyright Swisslog [IP AG], Switzerland. All rights reserved.
 * 
 * ------------------------------------------------------------------------------------
 *	
 * 	Revision History: 
 *
 * 	VERSION			DATE			INITIALS			DESCRIPTION
 *	0.1				01.01.2001		swl					Example
 *
 **************************************************************************************)


// Check reference is valid
IF __ISVALIDREF(SubsystemRegistry.rSubsystemData) THEN
	// Return subsystem data
	F_IsSubsystemInitialized := SubsystemRegistry.rSubsystemData.Init;
END_IF

END_FUNCTION

// ---- 20_Product/30_Toolbox/99_Misc/F_CreateHashCode.TcPOU
// returns the hash code from that given string
FUNCTION PUBLIC F_CreateHashCode : UDINT
(**************************************************************************************
 * 	Application		:	BoxControl Framework
 *	Revision		:	$Revision: 404529 $
 *	Revision date	:	$Date: 2018-04-23 08:21:38 +0200 (Mo., 23 Apr 2018) $
 *	Last changed by	:	$Author: b7bolm $
 *	URL				:	$URL: http://almscdc.swisslog.com/repo/SWPD/Development/BoxControlFramework/20_Release/trunk/01_Software/BCF/BCF/JumpStart/30_Toolbox/99_Misc/F_CreateHashCode.TcPOU $
 *
 *	Purpose			:	Creates a Hash code based on a string. This code only
 *						enhances the search algorithm - but is not a unique ID.
 *						A final check in comparison is always needed.
 *
 * ------------------------------------------------------------------------------------
 *	Copyright Swisslog [IP AG], Switzerland. All rights reserved.
 * 
 * ------------------------------------------------------------------------------------
 *	
 * 	Revision History: 
 *
 * 	VERSION			DATE			INITIALS			DESCRIPTION
 *	0.1				01.01.2001		swl					Example
 *
 **************************************************************************************)
VAR_INPUT
	InputString			: T_MaxString		:= '';		// String for creating the hash-code *)
END_VAR

VAR
	Result				: UDINT;
	Idx					: WORD;
END_VAR


// initializing
Result:= 0;
Idx   := 0;

// use every character to calculate
WHILE(InputString[Idx] <> 16#00)DO
	// calculate
	Result := (UDINT#19 * Result) + BYTE_TO_UDINT(InputString[Idx]);

	// next character
	Idx:= Idx + 1;
END_WHILE

// forward result
F_CreateHashCode:= Result;

END_FUNCTION

// ---- 20_Product/10_BCF/11_Conv/11_Com/11_ITC/F_ITC_SendGCR.TcPOU
FUNCTION F_ITC_SendGCR : BOOL
(**************************************************************************************
 * 	Application		:	BoxControl Framework
 *	Revision		:	$Revision: 404529 $
 *	Revision date	:	$Date: 2018-04-23 08:21:38 +0200 (Mo., 23 Apr 2018) $
 *	Last changed by	:	$Author: b7bolm $
 *	URL				:	$URL: http://almscdc.swisslog.com/repo/SWPD/Development/BoxControlFramework/20_Release/trunk/01_Software/BCF/BCF/JumpStart/20_Product/10_App/11_Com/10_Lib/10_Conv/11_ITC/F_ITC_SendGCR.TcPOU $
 *
 *	Purpose			:	Wrap message - GCR
 *
 * ------------------------------------------------------------------------------------
 *	Copyright Swisslog [IP AG], Switzerland. All rights reserved.
 * 
 * ------------------------------------------------------------------------------------
 *	
 * 	Revision History: 
 *
 * 	VERSION			DATE			INITIALS			DESCRIPTION
 *	0.1				01.01.2001		swl					Example
 *
 **************************************************************************************)
VAR_INPUT
	eChannelSrc		: E_MFCS_Channel; // Source communicaton channel	
	GroupName		: STRING(Conveyor.POSITION_STRINGLENGTH); // SIS Group Name MM-GGG-0000-000
	Code			: INT; // Control code
	Variable		: DINT; // Control code variable
	eReturnCode		: E_ErrorConv; // Return code
END_VAR
VAR
	GCR				: ST_ITC_GCR; 
END_VAR

// Map values
GCR.GroupName := GroupName;
GCR.Code := Code;
GCR.Variable := Variable;
GCR.ReturnCode := eReturnCode;

// Forward to ITC
F_ITC_SendGCR := fbITC_Manager.M_SendData(
					meChannel	:= eChannelSrc,
					mMsgType	:= E_ITC_MsgTypeConv.GROUP_CONTROL_REPLY,
					mpData		:= ADR(GCR),
					mLen		:= SIZEOF(GCR));

END_FUNCTION

// ---- 20_Product/10_BCF/11_Conv/11_Com/11_ITC/F_ITC_SendGSR.TcPOU
FUNCTION F_ITC_SendGSR : BOOL
(**************************************************************************************
 * 	Application		:	BoxControl Framework
 *	Revision		:	$Revision: 404529 $
 *	Revision date	:	$Date: 2018-04-23 08:21:38 +0200 (Mo., 23 Apr 2018) $
 *	Last changed by	:	$Author: b7bolm $
 *	URL				:	$URL: http://almscdc.swisslog.com/repo/SWPD/Development/BoxControlFramework/20_Release/trunk/01_Software/BCF/BCF/JumpStart/20_Product/10_App/11_Com/10_Lib/10_Conv/11_ITC/F_ITC_SendGSR.TcPOU $
 *
 *	Purpose			:	Wrap message - GSR
 *
 * ------------------------------------------------------------------------------------
 *	Copyright Swisslog [IP AG], Switzerland. All rights reserved.
 * 
 * ------------------------------------------------------------------------------------
 *	
 * 	Revision History: 
 *
 * 	VERSION			DATE			INITIALS			DESCRIPTION
 *	0.1				01.01.2001		swl					Example
 *
 **************************************************************************************)
VAR_INPUT
	eChannelSrc			: E_MFCS_Channel; // Source communicaton channel		
	GroupName			: STRING(Conveyor.POSITION_STRINGLENGTH); // SIS Group Name MM-GGG-0000-000
	eMode				: E_PositionMode; // Mode
	eState				: E_PositionState; // State
	eErrorState			: E_ErrorState; // Error State
	eErrorCode			: E_ErrorConv; // Return Code
	eErrorType			: E_ErrorType; // Error Type
	ErrorInformation	: STRING(System.ERROR_PARAM_STRINGLENGTH); // 5 Chars Error Information
	Variable			: DINT; // Variable
	eReturnCode			: E_ErrorConv; // Return code
END_VAR
VAR
	GSR					: ST_ITC_GSR; 
END_VAR

// Map values
GSR.GroupName := GroupName;
GSR.eState := eState;
GSR.eMode := eMode;
GSR.eErrorCode := eErrorCode;
GSR.eErrorState := eErrorState;
GSR.eErrorType := eErrorType;
GSR.ErrorInformation := ErrorInformation;
GSR.Variable := Variable;
GSR.eReturnCode := eReturnCode;

// Forward to ITC
F_ITC_SendGSR := fbITC_Manager.M_SendData(
					meChannel	:= eChannelSrc,
					mMsgType	:= E_ITC_MsgTypeConv.GROUP_STATUS_REPORT,
					mpData		:= ADR(GSR),
					mLen		:= SIZEOF(GSR));

END_FUNCTION

// ---- 20_Product/30_Toolbox/13_TimerCounter/FB_GeneratePulse.TcPOU
FUNCTION_BLOCK FB_GeneratePulse
(**************************************************************************************
 * 	Application		:	BoxControl Framework
 *	Revision		:	$Revision: 404529 $
 *	Revision date	:	$Date: 2018-04-23 08:21:38 +0200 (Mo., 23 Apr 2018) $
 *	Last changed by	:	$Author: b7bolm $
 *	URL				:	$URL: http://almscdc.swisslog.com/repo/SWPD/Development/BoxControlFramework/20_Release/trunk/01_Software/BCF/BCF/JumpStart/30_Toolbox/13_TimerCounter/FB_GeneratePulse.TcPOU $
 *
 *	Purpose			:	FB_GeneratePulse uses the internal sps timer to generate a continuous output waveform 
 *						with programmable high and low time. The accuracy of gen_pulse is depending on the task cycle time.
 *						Start = TRUE will start and Start = FALSE will stop the generator.The number of pulse can be 
 * 						preset with the "NumberOfPulses" Input. If "NumberOfPulses" is set to "0" then a continous waveform
 *      				is generated. The "Hold" input allows to stop the waveform at any point and continue the waveform at
 *     					the stop position after releasing the "Hold" input. The inputs "PulseTimeOn" and "PulseTimeOff" allows to 
 * 						to configure the waveform high and low time.
 *
 * ------------------------------------------------------------------------------------
 *	Copyright Swisslog [IP AG], Switzerland. All rights reserved.
 * 
 * ------------------------------------------------------------------------------------
 *	
 * 	Revision History: 
 *
 * 	VERSION			DATE			INITIALS			DESCRIPTION
 *	0.1				01.01.2001		swl					Example
 *
 **************************************************************************************)
VAR_INPUT
	Start		:BOOL;		(* Start Timer with rising edge, end puls generator with IN := FALSE *)
	Hold		:BOOL;		(* Hold generator with rising edge, continue timing with falling edge *)
	NumberOfPulses	:INT  := 0;	(* Number of expected pulses *)
	PulseTimeOn	:TIME := T#1S; (* Pulse time length for off puls *)
	PulseTimeOff	:TIME := T#1S; (* Pulse time length for on puls *)
END_VAR

VAR_OUTPUT
	Pulse		:BOOL;		(* Resulting puls *)
	eState		:E_PulsGen; (* Status for pulse generator *)
	CntPulses	:INT;		(* Actual count of generated pulses *)
END_VAR

VAR
	Init		:BOOL;		(* Initialize once timer with start trigger *)
	TimerOn		:FB_Timer;	(* Timer for on puls *)
	TimerOff	:FB_Timer;	(* Timer for off puls *)
END_VAR

IF Start THEN

	(* Check hold state *)
	IF NOT Hold THEN
		(* Run pulse sequence *)
		IF CntPulses < NumberOfPulses OR NumberOfPulses = 0 THEN
			(* Produce predefined number of pulses *)

			IF NOT Pulse THEN
				(* Timeout pulse off *)
				TimerOff(IN := TRUE, PT := PulseTimeOff, Hold := FALSE);

				(* If time elapsed or initializing then set pulse high *)
				IF TimerOff.Q OR NOT Init THEN
				 	Pulse := TRUE;
					TimerOff(IN := FALSE);
					TimerOn(IN := TRUE);
					Init := TRUE;
				END_IF
			ELSE
				(* Timeout pulse on *)
				TimerOn(IN := TRUE, PT := PulseTimeOn, hold := FALSE);

				(* If time elapsed set puls low *)
				IF TimerOn.Q THEN
				 	Pulse := FALSE;
					CntPulses := CntPulses + 1;
					TimerOn(IN := FALSE);
					TimerOff(IN := TRUE);
				END_IF
			END_IF
			eState := E_PulsGen.PG_BUSY;
		ELSE
			eState := E_PulsGen.PG_END;
		END_IF
	ELSE
		(* Pulse generator is on hold set timers on hold *)
		TimerOn(hold := TRUE);
		TimerOff(hold := TRUE);
	END_IF

ELSE
	(* Initialize values *)
	Init := FALSE;
	CntPulses := 0;
	eState := E_PulsGen.PG_READY;
	Pulse := FALSE;
	TimerOff(IN := FALSE);
	TimerOn(IN := FALSE);
END_IF

END_FUNCTION_BLOCK

// ---- 20_Product/30_Toolbox/13_TimerCounter/FB_Timer.TcPOU
FUNCTION_BLOCK FB_Timer
(**************************************************************************************
 * 	Application		:	BoxControl Framework
 *	Revision		:	$Revision: 404529 $
 *	Revision date	:	$Date: 2018-04-23 08:21:38 +0200 (Mo., 23 Apr 2018) $
 *	Last changed by	:	$Author: b7bolm $
 *	URL				:	$URL: http://almscdc.swisslog.com/repo/SWPD/Development/BoxControlFramework/20_Release/trunk/01_Software/BCF/BCF/JumpStart/30_Toolbox/13_TimerCounter/FB_Timer.TcPOU $
 *
 *	Purpose			:	This function allows to 
 *						A rising edge at the "Start" input causes a rising edge at output "TimeOut" 
 *						after the time PresetTime has expired. 
 *						A rising edge at the "Hold" input stops the timer. The timer continues after 
 *      				a falling edge at the "Hold" input.
 *      				The actual elapsed time is provided by the output "ElapsedTime"
 *
 * ------------------------------------------------------------------------------------
 *	Copyright Swisslog [IP AG], Switzerland. All rights reserved.
 * 
 * ------------------------------------------------------------------------------------
 *	
 * 	Revision History: 
 *
 * 	VERSION			DATE			INITIALS			DESCRIPTION
 *	0.1				01.01.2001		swl					Example
 *
 **************************************************************************************)
VAR_INPUT
	IN			:BOOL; (* Start Timer with rising edge*)
	Hold			:BOOL; (* Hold Timer with rising edge, continue timing with falling edge *)
	PT			:TIME; (* Time to pass, before Output "TimeOut" is set *)

END_VAR

VAR_OUTPUT
	Q			:BOOL; (* Time expired *)
    	ET 			:TIME; (* Time elapsed *)
END_VAR

VAR
	LastIN			:BOOL; (* Trigger detection for start signal *)
	LastHold		:BOOL; (* Trigger detection for hold signal *)
	StartTime		:TIME; (* Time stamp which is used to calculate the elapsed time *)
	HoldTime		:TIME; (* Time elapsed during the hold state *)
	StartHoldTime		:TIME; (* Time stamp which is used to calculate the hold time *)
END_VAR

IF IN THEN
	(* Detect start trigger an preset timer values at timer start *)
	IF NOT LastIN AND IN THEN
		startTime := TIME();
	END_IF

	(* Detect hold trigger and save actual time  *)
	IF NOT lastHold AND Hold  THEN
		StartHoldTime := TIME();
	END_IF

	(* Detect hold end trigger and move startTime by elapsed holdtime *)
	IF lastHold AND NOT hold THEN
		HoldTime := TIME() - StartHoldtime;
		startTime := startTime + HoldTime;
	END_IF

	IF NOT Hold AND NOT Q THEN
		(* Update elapsed time *)
		ET := TIME() - startTime;

		IF ET >= PT THEN
			Q := TRUE;
		ELSE
			Q := FALSE;
		END_IF
	END_IF

	LastHold  := Hold;

ELSE
	(* Initialize values *)
	ET 		:= T#0s;
	Q 		:= FALSE;
	StartTime	:= T#0s;
	HoldTime 	:= T#0s;
	StartHoldtime 	:= T#0s;
	LastIN		:= FALSE;
	LastHold	:= FALSE;
END_IF

LastIN := IN;

END_FUNCTION_BLOCK

// ---- 20_Product/10_BCF/11_Conv/10_Base/F_ResetError.TcPOU
FUNCTION F_ResetError : BOOL
(**************************************************************************************
 * 	Application		:	BoxControl Framework
 *	Revision		:	$Revision: 404529 $
 *	Revision date	:	$Date: 2018-04-23 08:21:38 +0200 (Mo., 23 Apr 2018) $
 *	Last changed by	:	$Author: b7bolm $
 *	URL				:	$URL: http://almscdc.swisslog.com/repo/SWPD/Development/BoxControlFramework/20_Release/trunk/01_Software/BCF/BCF/JumpStart/20_Product/10_App/10_Base/10_Lib/10_Conv/F_ResetError.TcPOU $
 *
 *	Purpose			:	Reset error
 *
 *
 * ------------------------------------------------------------------------------------
 *	Copyright Swisslog [IP AG], Switzerland. All rights reserved.
 * 
 * ------------------------------------------------------------------------------------
 *	
 * 	Revision History: 
 *
 * 	VERSION			DATE			INITIALS			DESCRIPTION
 *	0.1				01.01.2001		swl					Example
 *
 **************************************************************************************)
VAR_INPUT
	Reset		: BOOL; // Force reset
END_VAR

VAR_IN_OUT
	ErrorData	: ST_ErrorDataSet; // ErrorData of the moduls 
END_VAR

// Initialize
F_ResetError := FALSE;

// Reset error if ResetError command or reset command is set 
IF ErrorData.ResetError OR Reset THEN
	// Clear error
	ErrorData.ResetError 	:= FALSE; 
	ErrorData.ErrorType 	:= NO_ERROR_PENDING;
	ErrorData.ErrorCode.Conv:= E_ErrorConv.NO_ERROR_CODE;
	ErrorData.ErrorParam 	:= '';
	F_ResetError 			:= TRUE;
END_IF

END_FUNCTION

// ---- 20_Product/20_ProBox/22_ProMove/15_SubSystem/FB_ProBoxSubsystem.TcPOU
FUNCTION_BLOCK FB_ProBoxSubsystem EXTENDS FB_SubsystemConv
VAR_INPUT
	Config						: ST_CFG_ProBoxSubsystem; // Configuration 
	HW_Inputs					: ST_HW_InputsSubsystemManager; // Hardware inputs
END_VAR

VAR_OUTPUT
	HW_Outputs					: ST_HW_OutputsSubsystemManager; // Hardware outputs
	Outputs						: ST_OutputsSubsystemManager; // Outputs
END_VAR

VAR
	Inputs						: ST_InputsSubsystemManager; // Inputs
	EtherCatSupervision			: ARRAY [1..NUMBERS_OF_ETHERCAT_SLAVE_DIAG] OF ST_EtherCatDeviceStates; // EtherCAT supervision
	StopAllGroups				: BOOL; // Flag to stop all groups

	fbCpuUsage					: TC_CpuUsage; // Reads CPU usage 
	fbSysLatency				: TC_SysLatency; // Reads CPU latency 
	MaxCpuUsage 				: INT; // Max Cpu usage: [%] 
	
	CycleTime					: UDINT; // Cycle time of task: Time in [us] 
	ActExecutionTime			: UDINT; // Actual execution time of task: Time in [us] 
	MaxActExecutionTime     	: UDINT; // Maximum execution time of task: Time in [us] 

	fbUpdateSystemTime			: NT_SetLocalTime; // FB to set the RTC of th eIPC 
	LastSystemTimeUpdate		: DATE_AND_TIME; // TimeStamp of the last SystemTime update 
	UpdateSystemTime			: BOOL; // SystemTime update necessary 
	
	TimeSyncActive				: BOOL; // Time sync is active
	fbTimeReqReset				: TON; // Reset request after a certain time
	fbStoppingDelayTimer		: TON; // Delay stopping
	fbStartUpDelayTimer			: TON; // Timer delayed start up functions 
	
	Idx							: INT; // Iterator
	Name						: T_MaxString; // Name with alpha numeric signs only
	fbSystemInfo				: FB_SystemInfo; // Gathering system info
	fbGetCurTaskIdx  			: GETCURTASKINDEX; // Returns the actual task index	
	CpuUsageResetTimer			: TON :=(PT:=T#10S); // timer for reseting CPU usage error/warning
END_VAR

VAR PERSISTENT
	Settings					: ST_CFG_ProBoxSubsystem; // Settings
END_VAR


(**************************************************************************************************************
   Input mapping
***************************************************************************************************************)
A_InputMapping();


(**************************************************************************************************************
  Initialization
***************************************************************************************************************)
A_Init();


(**************************************************************************************************************
  Control system initialization
***************************************************************************************************************)
M_InitControl();


(**************************************************************************************************************
   Mode control
***************************************************************************************************************)
A_ModeControl();


(**************************************************************************************************************
   State control
***************************************************************************************************************)
A_StateControl();


(**************************************************************************************************************
 Subsystem monitoring
***************************************************************************************************************)
// Delay timer
fbStartUpDelayTimer(IN := SubsystemData.Init, PT := Settings.tDelayMonitoring);

// Wait until Subsystem is started up completely 
IF fbStartUpDelayTimer.Q THEN
	(**************************************************************************************************************
	   Monitor EtherCat master status
	***************************************************************************************************************)
	F_MonitorEtherCAT_Master(
		MasterDeviceState			:= UINT_TO_INT(HW_Inputs.EtherCAT_MasterState),
		MasterDeviceWorkingCounter	:= HW_Inputs.EtherCAT_MasterWorkingCounter,
		ErrorData					:= SubsystemData.ErrorData.ErrorDataSet[1]); 
		
		
	(**************************************************************************************************************
	   Monitor EtherCAT slaves
	***************************************************************************************************************)	
	A_SlaveDeviceSupervision();
	
	
	(**************************************************************************************************************
	   Monitor CPU states (temperature, fan)
	***************************************************************************************************************)
	A_MonitorCpuHardware();
	
	
	(**************************************************************************************************************
	   Monitor TwinCat (cpu usage, latency )
	***************************************************************************************************************)
	A_MonitorCpuUsage();
	
	
	(**************************************************************************************************************
	   Monitor MFCS connections (E.g. AM, SPOC)
	***************************************************************************************************************)
	A_MonitorMFCS_Connections();
END_IF


(**************************************************************************************************************
   Update SystemTime
***************************************************************************************************************)
A_UpdateSystemTime();


(**************************************************************************************************************
  Monitor subsystem errors
***************************************************************************************************************)
M_MonitorSubsystemErrors();


(**************************************************************************************************************
   ITC Handler Out
***************************************************************************************************************)
M_ITC_ProcessOut();


(**************************************************************************************************************
   Output mapping
***************************************************************************************************************)
A_OutputMapping();

ACTION A_Init:
// Update registry
M_UpdateRegistry();
 
// Set init-flag after one cycle 
IF NOT SubsystemData.Init AND SubsystemData.InitRunning THEN
	
	IF M_InitSubsystem(FALSE) THEN
		// Send status report - System restart
		ITC.Commands.SystemRestartInfo := TRUE;
	
		SubsystemData.Init := TRUE;
		SubsystemData.InitRunning := FALSE;
		
		// Set reset cmd
		SubsystemData.ErrorData.Error.ResetError := TRUE;
		
		// Print debug
		DebugMsg := CONCAT('Initialization done. Subsystem: ', SettingsSubsystem.SubsystemName);
		fbDebugMsg.M_SendInfoMsg(DebugMsg);
	END_IF
// If instance is not initialized
ELSIF NOT SubsystemData.Init THEN
	
	// Reset internal variables
	SubsystemData.OperationState := SubsystemBase.OperationStateEmpty;
	
	// Initialize values
	MaxActExecutionTime := 0;
	MaxCpuUsage := 0;
	UpdateSystemTime := FALSE;
	StopAllGroups := FALSE;
	CycleTime := 0;
	ActExecutionTime := 0;
	MaxActExecutionTime := 0;
	UpdateSystemTime := 0;
	TimeSyncActive := FALSE;
	SubsystemInterface.IN.MasterSpeed := 100;
	// Load configuration 
	Settings := Config;
	
	// Reset values and load config
	M_PreInit();
	
	// Init ongoing
	SubsystemData.InitRunning := TRUE;
END_IF
END_ACTION

ACTION A_InputMapping:
(**************************************************************************************
 * 	NAME		A_InputMapping
 * 	FUNCTION	Input mapping
 **************************************************************************************)
 
 
(**************************************************************************************************************
   HW input mapping
***************************************************************************************************************)

Inputs.EtherCAT_MasterState				:= HW_Inputs.EtherCAT_MasterState;
Inputs.EtherCAT_MasterWorkingCounter	:= HW_Inputs.EtherCAT_MasterWorkingCounter;
Inputs.DeviceState						:= HW_Inputs.DeviceState;

(**************************************************************************************************************
  Get system info
***************************************************************************************************************)
fbSystemInfo();

Inputs.CPU_Temperatur		:= fbSystemInfo.CPU_Temperatur;
Inputs.CPU_Usage			:= fbSystemInfo.CPU_Usage;
Inputs.SystemUsage			:= fbSystemInfo.SystemUsage;
Inputs.FanSpeed				:= fbSystemInfo.FanSpeed;
END_ACTION

ACTION A_ModeControl:
(**************************************************************************************
 * 	NAME		A_ModeControl
 * 	FUNCTION	Handle subsystem mode
 **************************************************************************************)
 
 // Subsystem mode
CASE SubSystemData.OperationState.eMode OF

	(*******************************************************************************
	  Unknown mode 
	********************************************************************************)
	E_PositionMode.UNKNOWN_MODE:
		// Switch to automated mode
		SubSystemData.OperationState.eMode := E_PositionMode.AUTO_MODE;
	
	(*******************************************************************************
	  Automatic mode
	********************************************************************************)
	E_PositionMode.AUTO_MODE:
		// Subsystem always in auto mode
		;
	
(********************************************************************************
	Error case
*********************************************************************************)
ELSE
	// Programming error
	DebugMsg := CONCAT(	'Programming error - Invalid SubSystem mode: ', 
					   	INT_TO_STRING(SubSystemData.OperationState.eMode));
		
	fbDebugMsg.M_SendErrorMsg(DebugMsg);
END_CASE
END_ACTION

ACTION A_MonitorCpuHardware:
(**************************************************************************************
 * 	NAME		A_MonitorCpuHardware
 * 	FUNCTION	Monitor the CPU as temperatures and fan speed
 *
 **************************************************************************************)

(**************************************************************************************
   Monitor CPU temperatur
***************************************************************************************)
// If cpu temperatur is under 80 °C
IF Inputs.CPU_Temperatur < Settings.CPU_TemperatureWarning THEN
	// Reset error
	F_ResetError(Reset := TRUE, ErrorData := SubSystemData.ErrorData.ErrorDataSet[3]);

// Warning > 85°C and < 95° C
ELSIF Inputs.CPU_Temperatur >= Settings.CPU_TemperatureWarning AND 
	  Inputs.CPU_Temperatur < Settings.CPU_TemperatureError THEN
	// Set warning
	F_SetError(	
		ErrorType	:= E_ErrorType.WARNING,
		ErrorParam	:= INT_TO_STRING(Inputs.CPU_Temperatur),
		ErrorMsg	:= E_ErrorConv.OVER_TEMPEREATURE_CPU,
		ErrorData	:= SubSystemData.ErrorData.ErrorDataSet[3]);
	
// Set error > 95°C
ELSIF Inputs.CPU_Temperatur >= Settings.CPU_TemperatureError THEN
	// Set error
	F_SetError(	
		ErrorType	:= E_ErrorType.ERROR,
		ErrorParam	:= INT_TO_STRING(Inputs.CPU_Temperatur),
		ErrorMsg	:= E_ErrorConv.OVER_TEMPEREATURE_CPU,
		ErrorData	:= SubSystemData.ErrorData.ErrorDataSet[3]);
END_IF

(**************************************************************************************
   Monitor Fan speed
***************************************************************************************)
// If fan is activated
IF Settings.CPU_FanExists THEN
	// Check fan speed
	IF Inputs.FanSpeed > Settings.MinFanSpeed THEN
		// Reset error
		F_ResetError(Reset := TRUE, ErrorData := SubSystemData.ErrorData.ErrorDataSet[4]);
	ELSE
		// Set error
		F_SetError(	
			ErrorType	:= E_ErrorType.ERROR,
			ErrorParam	:= UINT_TO_STRING(Inputs.FanSpeed),
			ErrorMsg	:= E_ErrorConv.FAN_ERROR_CPU,
			ErrorData	:= SubSystemData.ErrorData.ErrorDataSet[4]);
	END_IF
END_IF
END_ACTION

ACTION A_MonitorCpuUsage:
(**************************************************************************************
 * 	NAME		A_MonitorCpuUsage
 * 	FUNCTION	Monitor CPU usage
 *
 **************************************************************************************)

(**************************************************************************************
   CPU usage
***************************************************************************************)
// Reset error
CpuUsageResetTimer(IN:= (SubSystemData.ErrorData.ErrorDataSet[5].ErrorType = E_ErrorType.ERROR AND Inputs.CPU_Usage < Settings.CPU_UsageError) OR
						(SubSystemData.ErrorData.ErrorDataSet[5].ErrorType = E_ErrorType.WARNING AND Inputs.CPU_Usage < Settings.CPU_UsageWarning));

//reset error via SIS telegram or reset button
F_ResetError(
		Reset 		:= FALSE, 
		ErrorData 	:= SubSystemData.ErrorData.ErrorDataSet[5]);

//reset error automatically after 10 sec of no error / warning
IF(CpuUsageResetTimer.Q) THEN
	F_ResetError(
		Reset 		:= TRUE,
		ErrorData 	:= SubSystemData.ErrorData.ErrorDataSet[5]);
END_IF

// Track max Cpu usage 
IF Inputs.CPU_Usage > MaxCpuUsage THEN
	MaxCpuUsage := Inputs.CPU_Usage;
END_IF



IF(SubSystemData.ErrorData.ErrorDataSet[5].ErrorType <> E_ErrorType.ERROR)THEN

	// Usage > 60% and < 80%
	IF Inputs.CPU_Usage > Settings.CPU_UsageWarning AND Inputs.CPU_Usage < Settings.CPU_UsageError  THEN
		// Set warning
		F_SetError(	
			ErrorType	:= E_ErrorType.WARNING,
			ErrorParam	:= INT_TO_STRING(Inputs.CPU_Usage),
			ErrorMsg	:= E_ErrorConv.CPU_OVERLOAD,
			ErrorData	:= SubSystemData.ErrorData.ErrorDataSet[5]);
	
	// Usage > 80%
	ELSIF Inputs.CPU_Usage > Settings.CPU_UsageError THEN
		// Set error
		F_SetError(	
			ErrorType	:= E_ErrorType.ERROR,
			ErrorParam	:= INT_TO_STRING(Inputs.CPU_Usage),
			ErrorMsg	:= E_ErrorConv.CPU_OVERLOAD,
			ErrorData	:= SubSystemData.ErrorData.ErrorDataSet[5]);
	END_IF
END_IF

(**************************************************************************************
   System latency
***************************************************************************************)
// Get current task index
fbGetCurTaskIdx();

// Read cycle time [ms]
CycleTime :=  _TaskInfo[fbGetCurTaskIdx.index].CycleTime / 10;


// Read task time [ms]
ActExecutionTime :=  _TaskInfo[fbGetCurTaskIdx.index].LastExecTime / 10;

// Max actual execution [ms]
IF ActExecutionTime > MaxActExecutionTime THEN
	MaxActExecutionTime := ActExecutionTime;
END_IF
END_ACTION

ACTION A_MonitorMFCS_Connections:
(**************************************************************************************
 * 	NAME		A_MonitorTCPIP_Interface
 * 	FUNCTION	Monitor TCP-IP communication  
 **************************************************************************************)


(**************************************************************************************
   AM Connection
***************************************************************************************)
// If AM is configured
IF Settings.AM_Exists THEN
	
	// If AM is not connected
	IF NOT fbMFCS_Channel[E_MFCS_Channel.AM].M_IsConnected() THEN
		// Set error
		F_SetError(	
			ErrorType	:= E_ErrorType.ERROR,
			ErrorParam	:= '',
			ErrorMsg	:= E_ErrorConv.CONNECTION_ERROR_TO_AM,
			ErrorData	:= SubsystemData.ErrorData.ErrorDataSet[6]);
	ELSE
		// Reset error
		F_ResetError(Reset := TRUE, ErrorData := SubsystemData.ErrorData.ErrorDataSet[6]);
	END_IF
	
